LIN {X 0,Y 313.914,Z 800.321,A -85,B 0,C 180,E1 15407.149,E2 15407.149} C_VEL
LIN {X 0,Y 312.972,Z 809.816,A -85,B 0,C 180,E1 15404.241,E2 15404.241} C_VEL
LIN {X 0,Y 312.435,Z 817.558,A -85,B 0,C 180,E1 15401.257,E2 15401.257} C_VEL
LIN {X 0,Y 312.288,Z 823.487,A -85,B 0,C 180,E1 15398.284,E2 15398.284} C_VEL
LIN {X 0,Y 312.342,Z 827.951,A -85,B 0,C 180,E1 15395.143,E2 15395.143} C_VEL
LIN {X 0,Y 312.432,Z 830.624,A -85,B 0,C 180,E1 15392.017,E2 15392.017} C_VEL
LIN {X 0,Y 312.422,Z 831.58,A -85,B 0,C 180,E1 15389.083,E2 15389.083} C_VEL
LIN {X 0,Y 312.275,Z 830.966,A -85,B 0,C 180,E1 15385.961,E2 15385.961} C_VEL
LIN {X 0,Y 312.18,Z 828.719,A -85,B 0,C 180,E1 15382.824,E2 15382.824} C_VEL
LIN {X 0,Y 312.322,Z 824.551,A -85,B 0,C 180,E1 15379.486,E2 15379.486} C_VEL
LIN {X 0,Y 313.004,Z 818.517,A -85,B 0,C 180,E1 15376.138,E2 15376.138} C_VEL
LIN {X 0,Y 314.374,Z 810.506,A -85,B 0,C 180,E1 15372.795,E2 15372.795} C_VEL
LIN {X 0,Y 316.45,Z 800.994,A -85,B 0,C 180,E1 15369.662,E2 15369.662} C_VEL
LIN {X 0,Y 319.412,Z 789.139,A -85,B 0,C 180,E1 15366.517,E2 15366.517} C_VEL
LIN {X 0,Y 322.924,Z 776.215,A -85,B 0,C 180,E1 15363.719,E2 15363.719} C_VEL
LIN {X 0,Y 327.069,Z 761.596,A -85,B 0,C 180,E1 15361.118,E2 15361.118} C_VEL
LIN {X 0,Y 331.687,Z 745.535,A -85,B 0,C 180,E1 15358.769,E2 15358.769} C_VEL
LIN {X 0,Y 336.67,Z 727.913,A -85,B 0,C 180,E1 15356.672,E2 15356.672} C_VEL
LIN {X 0,Y 341.968,Z 708.641,A -85,B 0,C 180,E1 15354.83,E2 15354.83} C_VEL
LIN {X 0,Y 346.988,Z 689.431,A -85,B 0,C 180,E1 15353.382,E2 15353.382} C_VEL
LIN {X 0,Y 351.914,Z 668.887,A -85,B 0,C 180,E1 15352.194,E2 15352.194} C_VEL
LIN {X 0,Y 356.918,Z 643.713,A -85,B 0,C 180,E1 15351.101,E2 15351.101} C_VEL
LIN {X 0,Y 369.381,Z 576.188,A -85,B 0,C 180,E1 15348.561,E2 15348.561} C_VEL
LIN {X 0,Y 384.205,Z 508.645,A -85,B 0,C 180,E1 15346.075,E2 15346.075} C_VEL
LIN {X 0,Y 390.219,Z 483.209,A -85,B 0,C 180,E1 15344.294,E2 15344.294} C_VEL
LIN {X 0,Y 390.2,Z 483.501,A -85,B 0,C 180,E1 15343.942,E2 15343.942} C_VEL
LIN {X 0,Y 372.708,Z 558.454,A -85,B 0,C 180,E1 15341.257,E2 15341.257} C_VEL
LIN {X 0,Y 359.717,Z 624.486,A -85,B 0,C 180,E1 15338.782,E2 15338.782} C_VEL
LIN {X 0,Y 355.652,Z 646.636,A -85,B 0,C 180,E1 15337.785,E2 15337.785} C_VEL
LIN {X 0,Y 351.441,Z 666.051,A -85,B 0,C 180,E1 15336.586,E2 15336.586} C_VEL
LIN {X 0,Y 346.839,Z 684.676,A -85,B 0,C 180,E1 15335.107,E2 15335.107} C_VEL
LIN {X 0,Y 341.835,Z 703.189,A -85,B 0,C 180,E1 15333.259,E2 15333.259} C_VEL
LIN {X 0,Y 336.939,Z 719.84,A -85,B 0,C 180,E1 15331.186,E2 15331.186} C_VEL
LIN {X 0,Y 331.947,Z 735.894,A -85,B 0,C 180,E1 15328.713,E2 15328.713} C_VEL
LIN {X 0,Y 327.477,Z 749.759,A -85,B 0,C 180,E1 15326.082,E2 15326.082} C_VEL
LIN {X 0,Y 323.543,Z 761.616,A -85,B 0,C 180,E1 15323.301,E2 15323.301} C_VEL
LIN {X 0,Y 320.106,Z 771.924,A -85,B 0,C 180,E1 15320.286,E2 15320.286} C_VEL
LIN {X 0,Y 317.4,Z 780.232,A -85,B 0,C 180,E1 15317.224,E2 15317.224} C_VEL
LIN {X 0,Y 315.273,Z 787.058,A -85,B 0,C 180,E1 15313.947,E2 15313.947} C_VEL
LIN {X 0,Y 313.823,Z 792.027,A -85,B 0,C 180,E1 15310.649,E2 15310.649} C_VEL
LIN {X 0,Y 312.936,Z 795.242,A -85,B 0,C 180,E1 15307.342,E2 15307.342} C_VEL
LIN {X 0,Y 312.466,Z 796.765,A -85,B 0,C 180,E1 15304.037,E2 15304.037} C_VEL
LIN {X 0,Y 312.272,Z 796.643,A -85,B 0,C 180,E1 15300.917,E2 15300.917} C_VEL
LIN {X 0,Y 312.209,Z 794.933,A -85,B 0,C 180,E1 15297.704,E2 15297.704} C_VEL
LIN {X 0,Y 312.292,Z 791.564,A -85,B 0,C 180,E1 15294.488,E2 15294.488} C_VEL
LIN {X 0,Y 312.576,Z 786.605,A -85,B 0,C 180,E1 15291.353,E2 15291.353} C_VEL
LIN {X 0,Y 313.171,Z 779.862,A -85,B 0,C 180,E1 15288.209,E2 15288.209} C_VEL
LIN {X 0,Y 314.108,Z 771.702,A -85,B 0,C 180,E1 15285.247,E2 15285.247} C_VEL
LIN {X 0,Y 315.49,Z 761.548,A -85,B 0,C 180,E1 15282.287,E2 15282.287} C_VEL
LIN {X 0,Y 317.239,Z 749.878,A -85,B 0,C 180,E1 15279.522,E2 15279.522} C_VEL
LIN {X 0,Y 319.384,Z 736.161,A -85,B 0,C 180,E1 15276.865,E2 15276.865} C_VEL
LIN {X 0,Y 321.708,Z 721.337,A -85,B 0,C 180,E1 15274.503,E2 15274.503} C_VEL
LIN {X 0,Y 324.195,Z 704.826,A -85,B 0,C 180,E1 15272.344,E2 15272.344} C_VEL
LIN {X 0,Y 326.663,Z 687.236,A -85,B 0,C 180,E1 15270.475,E2 15270.475} C_VEL
LIN {X 0,Y 328.922,Z 669.075,A -85,B 0,C 180,E1 15268.94,E2 15268.94} C_VEL
LIN {X 0,Y 330.927,Z 649.75,A -85,B 0,C 180,E1 15267.67,E2 15267.67} C_VEL
LIN {X 0,Y 332.636,Z 629.153,A -85,B 0,C 180,E1 15266.675,E2 15266.675} C_VEL
LIN {X 0,Y 334.014,Z 605.352,A -85,B 0,C 180,E1 15265.907,E2 15265.907} C_VEL
LIN {X 0,Y 342.851,Z 452.576,A -85,B 0,C 180,E1 15261.576,E2 15261.576} C_VEL
LIN {X 0,Y 328.485,Z 422.487,A -85,B 0,C 180,E1 15259.015,E2 15259.015} C_VEL
LIN {X 0,Y 324.144,Z 413.761,A -85,B 0,C 180,E1 15258.154,E2 15258.154} C_VEL
LIN {X 0,Y 316.77,Z 394.569,A -85,B 0,C 180,E1 15254.74,E2 15254.74} C_VEL
LIN {X 0,Y 314.112,Z 387.671,A -85,B 0,C 180,E1 15253.437,E2 15253.437} C_VEL
LIN {X 0,Y 314.116,Z 387.671,A -85,B 0,C 180,E1 15249.042,E2 15249.042} C_VEL
LIN {X 0,Y 314.129,Z 387.672,A -85,B 0,C 180,E1 15244.733,E2 15244.733} C_VEL
LIN {X 0,Y 314.151,Z 387.67,A -85,B 0,C 180,E1 15240.399,E2 15240.399} C_VEL
LIN {X 0,Y 314.137,Z 387.667,A -85,B 0,C 180,E1 15236.055,E2 15236.055} C_VEL
LIN {X 0,Y 314.122,Z 387.667,A -85,B 0,C 180,E1 15231.651,E2 15231.651} C_VEL
LIN {X 0,Y 314.112,Z 387.664,A -85,B 0,C 180,E1 15227.219,E2 15227.219} C_VEL
LIN {X 0,Y 314.11,Z 387.664,A -85,B 0,C 180,E1 15222.875,E2 15222.875} C_VEL
LIN {X 0,Y 314.128,Z 387.662,A -85,B 0,C 180,E1 15218.419,E2 15218.419} C_VEL
LIN {X 0,Y 314.137,Z 387.66,A -85,B 0,C 180,E1 15214.015,E2 15214.015} C_VEL
LIN {X 0,Y 314.13,Z 387.664,A -85,B 0,C 180,E1 15209.635,E2 15209.635} C_VEL
LIN {X 0,Y 314.112,Z 387.669,A -85,B 0,C 180,E1 15205.253,E2 15205.253} C_VEL
LIN {X 0,Y 314.108,Z 387.668,A -85,B 0,C 180,E1 15200.842,E2 15200.842} C_VEL
LIN {X 0,Y 314.117,Z 387.667,A -85,B 0,C 180,E1 15196.376,E2 15196.376} C_VEL
LIN {X 0,Y 314.133,Z 387.668,A -85,B 0,C 180,E1 15192.016,E2 15192.016} C_VEL
LIN {X 0,Y 314.143,Z 387.669,A -85,B 0,C 180,E1 15187.546,E2 15187.546} C_VEL
LIN {X 0,Y 314.115,Z 387.668,A -85,B 0,C 180,E1 15183.034,E2 15183.034} C_VEL
LIN {X 0,Y 314.109,Z 387.672,A -85,B 0,C 180,E1 15178.531,E2 15178.531} C_VEL
LIN {X 0,Y 314.116,Z 387.676,A -85,B 0,C 180,E1 15174.148,E2 15174.148} C_VEL
LIN {X 0,Y 314.135,Z 387.67,A -85,B 0,C 180,E1 15169.749,E2 15169.749} C_VEL
LIN {X 0,Y 314.134,Z 387.669,A -85,B 0,C 180,E1 15165.297,E2 15165.297} C_VEL
LIN {X 0,Y 313.812,Z 388.707,A -85,B 0,C 180,E1 15164.32,E2 15164.32} C_VEL
LIN {X 0,Y 312.995,Z 391.85,A -85,B 0,C 180,E1 15163.251,E2 15163.251} C_VEL
LIN {X 0,Y 311.72,Z 398.473,A -85,B 0,C 180,E1 15161.831,E2 15161.831} C_VEL
LIN {X 0,Y 311.345,Z 405.44,A -85,B 0,C 180,E1 15160.402,E2 15160.402} C_VEL
LIN {X 0,Y 311.719,Z 407.553,A -85,B 0,C 180,E1 15159.912,E2 15159.912} C_VEL
LIN {X 0,Y 316.265,Z 424.463,A -85,B 0,C 180,E1 15155.968,E2 15155.968} C_VEL
LIN {X 0,Y 319.293,Z 436.92,A -85,B 0,C 180,E1 15153.231,E2 15153.231} C_VEL
LIN {X 0,Y 315.46,Z 463.796,A -85,B 0,C 180,E1 15148.388,E2 15148.388} C_VEL
LIN {X 0,Y 313.788,Z 477.545,A -85,B 0,C 180,E1 15145.985,E2 15145.985} C_VEL
LIN {X 0,Y 317.652,Z 514.782,A -85,B 0,C 180,E1 15144.352,E2 15144.352} C_VEL
LIN {X 0,Y 313.153,Z 610.478,A -85,B 0,C 180,E1 15141.066,E2 15141.066} C_VEL
LIN {X 0,Y 312.346,Z 627.663,A -85,B 0,C 180,E1 15140.142,E2 15140.142} C_VEL
LIN {X 0,Y 311.341,Z 644.035,A -85,B 0,C 180,E1 15138.927,E2 15138.927} C_VEL
LIN {X 0,Y 310.15,Z 660.173,A -85,B 0,C 180,E1 15137.35,E2 15137.35} C_VEL
LIN {X 0,Y 309.02,Z 675.002,A -85,B 0,C 180,E1 15135.482,E2 15135.482} C_VEL
LIN {X 0,Y 307.953,Z 688.503,A -85,B 0,C 180,E1 15133.328,E2 15133.328} C_VEL
LIN {X 0,Y 307.115,Z 699.77,A -85,B 0,C 180,E1 15131.075,E2 15131.075} C_VEL
LIN {X 0,Y 306.548,Z 709.041,A -85,B 0,C 180,E1 15128.776,E2 15128.776} C_VEL
LIN {X 0,Y 306.169,Z 717.713,A -85,B 0,C 180,E1 15125.999,E2 15125.999} C_VEL
LIN {X 0,Y 306.109,Z 723.767,A -85,B 0,C 180,E1 15123.371,E2 15123.371} C_VEL
LIN {X 0,Y 306.331,Z 728.031,A -85,B 0,C 180,E1 15120.748,E2 15120.748} C_VEL
LIN {X 0,Y 306.844,Z 730.658,A -85,B 0,C 180,E1 15117.946,E2 15117.946} C_VEL
LIN {X 0,Y 307.658,Z 731.453,A -85,B 0,C 180,E1 15115.34,E2 15115.34} C_VEL
LIN {X 0,Y 308.807,Z 730.568,A -85,B 0,C 180,E1 15112.746,E2 15112.746} C_VEL
LIN {X 0,Y 310.49,Z 727.787,A -85,B 0,C 180,E1 15109.986,E2 15109.986} C_VEL
LIN {X 0,Y 312.493,Z 723.453,A -85,B 0,C 180,E1 15107.434,E2 15107.434} C_VEL
LIN {X 0,Y 315.283,Z 716.356,A -85,B 0,C 180,E1 15104.598,E2 15104.598} C_VEL
LIN {X 0,Y 318.084,Z 708.328,A -85,B 0,C 180,E1 15102.248,E2 15102.248} C_VEL
LIN {X 0,Y 321.279,Z 698.442,A -85,B 0,C 180,E1 15099.981,E2 15099.981} C_VEL
LIN {X 0,Y 325.031,Z 685.498,A -85,B 0,C 180,E1 15097.672,E2 15097.672} C_VEL
LIN {X 0,Y 328.663,Z 671.745,A -85,B 0,C 180,E1 15095.752,E2 15095.752} C_VEL
LIN {X 0,Y 332.541,Z 655.405,A -85,B 0,C 180,E1 15093.961,E2 15093.961} C_VEL
LIN {X 0,Y 335.996,Z 638.369,A -85,B 0,C 180,E1 15092.532,E2 15092.532} C_VEL
LIN {X 0,Y 338.941,Z 621.261,A -85,B 0,C 180,E1 15091.452,E2 15091.452} C_VEL
LIN {X 0,Y 348.284,Z 567.539,A -85,B 0,C 180,E1 15088.946,E2 15088.946} C_VEL
LIN {X 0,Y 355.162,Z 531.054,A -85,B 0,C 180,E1 15087.337,E2 15087.337} C_VEL
LIN {X 0,Y 355.87,Z 516.287,A -85,B 0,C 180,E1 15085.732,E2 15085.732} C_VEL
LIN {X 0,Y 356.726,Z 501.332,A -85,B 0,C 180,E1 15083.743,E2 15083.743} C_VEL
LIN {X 0,Y 357.866,Z 489.179,A -85,B 0,C 180,E1 15081.767,E2 15081.767} C_VEL
LIN {X 0,Y 357.74,Z 486,A -85,B 0,C 180,E1 15079.731,E2 15079.731} C_VEL
LIN {X 0,Y 358.151,Z 485.015,A -85,B 0,C 180,E1 15078.147,E2 15078.147} C_VEL
LIN {X 0,Y 359.009,Z 484.902,A -85,B 0,C 180,E1 15076.755,E2 15076.755} C_VEL
LIN {X 0,Y 361.058,Z 488.224,A -85,B 0,C 180,E1 15074.401,E2 15074.401} C_VEL
LIN {X 0,Y 361.187,Z 488.98,A -85,B 0,C 180,E1 15074.208,E2 15074.208} C_VEL
LIN {X 0,Y 360.176,Z 501.484,A -85,B 0,C 180,E1 15073.084,E2 15073.084} C_VEL
LIN {X 0,Y 359.266,Z 508.394,A -85,B 0,C 180,E1 15072.71,E2 15072.71} C_VEL
LIN {X 0,Y 347.71,Z 581.363,A -85,B 0,C 180,E1 15070.114,E2 15070.114} C_VEL
LIN {X 0,Y 338.375,Z 654.777,A -85,B 0,C 180,E1 15067.523,E2 15067.523} C_VEL
LIN {X 0,Y 334.909,Z 673.937,A -85,B 0,C 180,E1 15066.556,E2 15066.556} C_VEL
LIN {X 0,Y 330.768,Z 692.92,A -85,B 0,C 180,E1 15065.266,E2 15065.266} C_VEL
LIN {X 0,Y 326.424,Z 710.758,A -85,B 0,C 180,E1 15063.671,E2 15063.671} C_VEL
LIN {X 0,Y 322.018,Z 727.541,A -85,B 0,C 180,E1 15061.756,E2 15061.756} C_VEL
LIN {X 0,Y 317.756,Z 743.428,A -85,B 0,C 180,E1 15059.502,E2 15059.502} C_VEL
LIN {X 0,Y 313.809,Z 758.314,A -85,B 0,C 180,E1 15056.901,E2 15056.901} C_VEL
LIN {X 0,Y 310.363,Z 771.95,A -85,B 0,C 180,E1 15053.949,E2 15053.949} C_VEL
LIN {X 0,Y 308.809,Z 779.29,A -85,B 0,C 180,E1 15052.179,E2 15052.179} C_VEL
LIN {X 0,Y 306.989,Z 791.913,A -85,B 0,C 180,E1 15049.403,E2 15049.403} C_VEL
LIN {X 0,Y 305.657,Z 802.566,A -85,B 0,C 180,E1 15046.535,E2 15046.535} C_VEL
LIN {X 0,Y 304.796,Z 811.742,A -85,B 0,C 180,E1 15043.469,E2 15043.469} C_VEL
LIN {X 0,Y 304.374,Z 818.957,A -85,B 0,C 180,E1 15040.409,E2 15040.409} C_VEL
LIN {X 0,Y 304.315,Z 824.411,A -85,B 0,C 180,E1 15037.362,E2 15037.362} C_VEL
LIN {X 0,Y 304.39,Z 828.204,A -85,B 0,C 180,E1 15034.333,E2 15034.333} C_VEL
LIN {X 0,Y 304.467,Z 830.382,A -85,B 0,C 180,E1 15031.317,E2 15031.317} C_VEL
LIN {X 0,Y 304.405,Z 831.05,A -85,B 0,C 180,E1 15028.306,E2 15028.306} C_VEL
LIN {X 0,Y 304.246,Z 830.152,A -85,B 0,C 180,E1 15025.098,E2 15025.098} C_VEL
LIN {X 0,Y 304.181,Z 827.428,A -85,B 0,C 180,E1 15021.684,E2 15021.684} C_VEL
LIN {X 0,Y 304.497,Z 822.9,A -85,B 0,C 180,E1 15018.253,E2 15018.253} C_VEL
LIN {X 0,Y 305.457,Z 816.503,A -85,B 0,C 180,E1 15014.819,E2 15014.819} C_VEL
LIN {X 0,Y 307.204,Z 808.16,A -85,B 0,C 180,E1 15011.4,E2 15011.4} C_VEL
LIN {X 0,Y 309.712,Z 798.308,A -85,B 0,C 180,E1 15008.206,E2 15008.206} C_VEL
LIN {X 0,Y 313.115,Z 786.372,A -85,B 0,C 180,E1 15005.07,E2 15005.07} C_VEL
LIN {X 0,Y 317.214,Z 772.901,A -85,B 0,C 180,E1 15002.193,E2 15002.193} C_VEL
LIN {X 0,Y 322.052,Z 757.414,A -85,B 0,C 180,E1 14999.495,E2 14999.495} C_VEL
LIN {X 0,Y 327.431,Z 740.36,A -85,B 0,C 180,E1 14997.074,E2 14997.074} C_VEL
LIN {X 0,Y 333.036,Z 722.382,A -85,B 0,C 180,E1 14995.01,E2 14995.01} C_VEL
LIN {X 0,Y 338.673,Z 703.62,A -85,B 0,C 180,E1 14993.285,E2 14993.285} C_VEL
LIN {X 0,Y 344.197,Z 684.057,A -85,B 0,C 180,E1 14991.881,E2 14991.881} C_VEL
LIN {X 0,Y 349.702,Z 662.484,A -85,B 0,C 180,E1 14990.705,E2 14990.705} C_VEL
LIN {X 0,Y 354.983,Z 637.145,A -85,B 0,C 180,E1 14989.648,E2 14989.648} C_VEL
LIN {X 0,Y 369.06,Z 569.328,A -85,B 0,C 180,E1 14987.076,E2 14987.076} C_VEL
LIN {X 0,Y 383.069,Z 510.953,A -85,B 0,C 180,E1 14984.941,E2 14984.941} C_VEL
LIN {X 0,Y 384.903,Z 503.746,A -85,B 0,C 180,E1 14984.433,E2 14984.433} C_VEL
LIN {X 0,Y 366.246,Z 580.486,A -85,B 0,C 180,E1 14981.677,E2 14981.677} C_VEL
LIN {X 0,Y 353.953,Z 639.883,A -85,B 0,C 180,E1 14979.346,E2 14979.346} C_VEL
LIN {X 0,Y 349.545,Z 659.245,A -85,B 0,C 180,E1 14978.264,E2 14978.264} C_VEL
LIN {X 0,Y 344.428,Z 678.747,A -85,B 0,C 180,E1 14976.831,E2 14976.831} C_VEL
LIN {X 0,Y 339.078,Z 697.275,A -85,B 0,C 180,E1 14975.1,E2 14975.1} C_VEL
LIN {X 0,Y 333.777,Z 714.058,A -85,B 0,C 180,E1 14973.14,E2 14973.14} C_VEL
LIN {X 0,Y 328.29,Z 730.451,A -85,B 0,C 180,E1 14970.775,E2 14970.775} C_VEL
LIN {X 0,Y 323.311,Z 744.731,A -85,B 0,C 180,E1 14968.24,E2 14968.24} C_VEL
LIN {X 0,Y 318.706,Z 757.419,A -85,B 0,C 180,E1 14965.455,E2 14965.455} C_VEL
LIN {X 0,Y 314.609,Z 768.541,A -85,B 0,C 180,E1 14962.418,E2 14962.418} C_VEL
LIN {X 0,Y 311.122,Z 778.117,A -85,B 0,C 180,E1 14959.119,E2 14959.119} C_VEL
LIN {X 0,Y 308.492,Z 785.539,A -85,B 0,C 180,E1 14955.798,E2 14955.798} C_VEL
LIN {X 0,Y 306.613,Z 791.116,A -85,B 0,C 180,E1 14952.428,E2 14952.428} C_VEL
LIN {X 0,Y 305.336,Z 795.076,A -85,B 0,C 180,E1 14948.853,E2 14948.853} C_VEL
LIN {X 0,Y 304.656,Z 797.074,A -85,B 0,C 180,E1 14945.461,E2 14945.461} C_VEL
LIN {X 0,Y 304.338,Z 797.395,A -85,B 0,C 180,E1 14942.071,E2 14942.071} C_VEL
LIN {X 0,Y 304.23,Z 796.153,A -85,B 0,C 180,E1 14938.87,E2 14938.87} C_VEL
LIN {X 0,Y 304.248,Z 793.36,A -85,B 0,C 180,E1 14935.665,E2 14935.665} C_VEL
LIN {X 0,Y 304.478,Z 788.598,A -85,B 0,C 180,E1 14932.262,E2 14932.262} C_VEL
LIN {X 0,Y 304.983,Z 782.305,A -85,B 0,C 180,E1 14929.038,E2 14929.038} C_VEL
LIN {X 0,Y 305.824,Z 774.628,A -85,B 0,C 180,E1 14925.999,E2 14925.999} C_VEL
LIN {X 0,Y 307.107,Z 765.001,A -85,B 0,C 180,E1 14922.961,E2 14922.961} C_VEL
LIN {X 0,Y 308.767,Z 753.934,A -85,B 0,C 180,E1 14920.122,E2 14920.122} C_VEL
LIN {X 0,Y 310.92,Z 740.503,A -85,B 0,C 180,E1 14917.3,E2 14917.3} C_VEL
LIN {X 0,Y 313.294,Z 725.893,A -85,B 0,C 180,E1 14914.782,E2 14914.782} C_VEL
LIN {X 0,Y 315.782,Z 710.168,A -85,B 0,C 180,E1 14912.558,E2 14912.558} C_VEL
LIN {X 0,Y 318.316,Z 692.905,A -85,B 0,C 180,E1 14910.574,E2 14910.574} C_VEL
LIN {X 0,Y 320.811,Z 674.138,A -85,B 0,C 180,E1 14908.844,E2 14908.844} C_VEL
LIN {X 0,Y 322.921,Z 655.67,A -85,B 0,C 180,E1 14907.506,E2 14907.506} C_VEL
LIN {X 0,Y 324.788,Z 635.515,A -85,B 0,C 180,E1 14906.402,E2 14906.402} C_VEL
LIN {X 0,Y 326.212,Z 614.334,A -85,B 0,C 180,E1 14905.609,E2 14905.609} C_VEL
LIN {X 0,Y 335.81,Z 455.019,A -85,B 0,C 180,E1 14900.964,E2 14900.964} C_VEL
LIN {X 0,Y 322.329,Z 426.659,A -85,B 0,C 180,E1 14898.482,E2 14898.482} C_VEL
LIN {X 0,Y 316.044,Z 414.082,A -85,B 0,C 180,E1 14897.221,E2 14897.221} C_VEL
LIN {X 0,Y 308.675,Z 395.185,A -85,B 0,C 180,E1 14893.752,E2 14893.752} C_VEL
LIN {X 0,Y 306.203,Z 388.657,A -85,B 0,C 180,E1 14892.526,E2 14892.526} C_VEL
LIN {X 0,Y 306.198,Z 388.656,A -85,B 0,C 180,E1 14888.097,E2 14888.097} C_VEL
LIN {X 0,Y 306.179,Z 388.661,A -85,B 0,C 180,E1 14883.619,E2 14883.619} C_VEL
LIN {X 0,Y 306.172,Z 388.657,A -85,B 0,C 180,E1 14879.117,E2 14879.117} C_VEL
LIN {X 0,Y 306.187,Z 388.658,A -85,B 0,C 180,E1 14874.708,E2 14874.708} C_VEL
LIN {X 0,Y 306.204,Z 388.653,A -85,B 0,C 180,E1 14870.251,E2 14870.251} C_VEL
LIN {X 0,Y 306.188,Z 388.661,A -85,B 0,C 180,E1 14865.726,E2 14865.726} C_VEL
LIN {X 0,Y 306.173,Z 388.66,A -85,B 0,C 180,E1 14861.3,E2 14861.3} C_VEL
LIN {X 0,Y 306.175,Z 388.657,A -85,B 0,C 180,E1 14856.752,E2 14856.752} C_VEL
LIN {X 0,Y 306.192,Z 388.652,A -85,B 0,C 180,E1 14852.236,E2 14852.236} C_VEL
LIN {X 0,Y 306.199,Z 388.646,A -85,B 0,C 180,E1 14847.941,E2 14847.941} C_VEL
LIN {X 0,Y 306.182,Z 388.653,A -85,B 0,C 180,E1 14843.437,E2 14843.437} C_VEL
LIN {X 0,Y 306.17,Z 388.658,A -85,B 0,C 180,E1 14838.891,E2 14838.891} C_VEL
LIN {X 0,Y 306.173,Z 388.661,A -85,B 0,C 180,E1 14834.446,E2 14834.446} C_VEL
LIN {X 0,Y 306.197,Z 388.658,A -85,B 0,C 180,E1 14829.948,E2 14829.948} C_VEL
LIN {X 0,Y 306.196,Z 388.655,A -85,B 0,C 180,E1 14825.499,E2 14825.499} C_VEL
LIN {X 0,Y 306.179,Z 388.657,A -85,B 0,C 180,E1 14821.067,E2 14821.067} C_VEL
LIN {X 0,Y 306.17,Z 388.664,A -85,B 0,C 180,E1 14816.502,E2 14816.502} C_VEL
LIN {X 0,Y 306.176,Z 388.664,A -85,B 0,C 180,E1 14812.125,E2 14812.125} C_VEL
LIN {X 0,Y 306.197,Z 388.658,A -85,B 0,C 180,E1 14807.726,E2 14807.726} C_VEL
LIN {X 0,Y 306.196,Z 388.85,A -85,B 0,C 180,E1 14804.613,E2 14804.613} C_VEL
LIN {X 0,Y 311.185,Z 405.516,A -85,B 0,C 180,E1 14800.403,E2 14800.403} C_VEL
LIN {X 0,Y 311.719,Z 407.553,A -85,B 0,C 180,E1 14799.912,E2 14799.912} C_VEL
LIN {X 0,Y 312.041,Z 412.58,A -85,B 0,C 180,E1 14798.827,E2 14798.827} C_VEL
LIN {X 0,Y 309.592,Z 428.14,A -85,B 0,C 180,E1 14795.884,E2 14795.884} C_VEL
LIN {X 0,Y 309.952,Z 431.807,A -85,B 0,C 180,E1 14795.106,E2 14795.106} C_VEL
LIN {X 0,Y 311.591,Z 439.271,A -85,B 0,C 180,E1 14793.455,E2 14793.455} C_VEL
LIN {X 0,Y 307.589,Z 466.366,A -85,B 0,C 180,E1 14788.478,E2 14788.478} C_VEL
LIN {X 0,Y 306.18,Z 477.362,A -85,B 0,C 180,E1 14786.52,E2 14786.52} C_VEL
LIN {X 0,Y 310.041,Z 515.528,A -85,B 0,C 180,E1 14784.8,E2 14784.8} C_VEL
LIN {X 0,Y 305.377,Z 611.092,A -85,B 0,C 180,E1 14781.406,E2 14781.406} C_VEL
LIN {X 0,Y 304.546,Z 628.058,A -85,B 0,C 180,E1 14780.466,E2 14780.466} C_VEL
LIN {X 0,Y 303.441,Z 645.323,A -85,B 0,C 180,E1 14779.139,E2 14779.139} C_VEL
LIN {X 0,Y 302.217,Z 661.31,A -85,B 0,C 180,E1 14777.522,E2 14777.522} C_VEL
LIN {X 0,Y 301.013,Z 676.765,A -85,B 0,C 180,E1 14775.509,E2 14775.509} C_VEL
LIN {X 0,Y 299.899,Z 690.654,A -85,B 0,C 180,E1 14773.212,E2 14773.212} C_VEL
LIN {X 0,Y 299.048,Z 702.238,A -85,B 0,C 180,E1 14770.792,E2 14770.792} C_VEL
LIN {X 0,Y 298.478,Z 711.743,A -85,B 0,C 180,E1 14768.282,E2 14768.282} C_VEL
LIN {X 0,Y 298.191,Z 719.199,A -85,B 0,C 180,E1 14765.774,E2 14765.774} C_VEL
LIN {X 0,Y 298.179,Z 725.59,A -85,B 0,C 180,E1 14762.883,E2 14762.883} C_VEL
LIN {X 0,Y 298.46,Z 729.696,A -85,B 0,C 180,E1 14760.192,E2 14760.192} C_VEL
LIN {X 0,Y 299.104,Z 732.227,A -85,B 0,C 180,E1 14757.318,E2 14757.318} C_VEL
LIN {X 0,Y 300.046,Z 732.895,A -85,B 0,C 180,E1 14754.646,E2 14754.646} C_VEL
LIN {X 0,Y 301.605,Z 731.64,A -85,B 0,C 180,E1 14751.613,E2 14751.613} C_VEL
LIN {X 0,Y 303.429,Z 728.808,A -85,B 0,C 180,E1 14748.982,E2 14748.982} C_VEL
LIN {X 0,Y 306.068,Z 723.475,A -85,B 0,C 180,E1 14746.011,E2 14746.011} C_VEL
LIN {X 0,Y 308.888,Z 716.782,A -85,B 0,C 180,E1 14743.45,E2 14743.45} C_VEL
LIN {X 0,Y 312.242,Z 708.123,A -85,B 0,C 180,E1 14740.936,E2 14740.936} C_VEL
LIN {X 0,Y 316.092,Z 697.002,A -85,B 0,C 180,E1 14738.474,E2 14738.474} C_VEL
LIN {X 0,Y 319.791,Z 685.109,A -85,B 0,C 180,E1 14736.409,E2 14736.409} C_VEL
LIN {X 0,Y 323.633,Z 671.93,A -85,B 0,C 180,E1 14734.568,E2 14734.568} C_VEL
LIN {X 0,Y 327.842,Z 655.543,A -85,B 0,C 180,E1 14732.776,E2 14732.776} C_VEL
LIN {X 0,Y 331.607,Z 638.669,A -85,B 0,C 180,E1 14731.353,E2 14731.353} C_VEL
LIN {X 0,Y 334.979,Z 620.426,A -85,B 0,C 180,E1 14730.212,E2 14730.212} C_VEL
LIN {X 0,Y 349.202,Z 546.392,A -85,B 0,C 180,E1 14726.798,E2 14726.798} C_VEL
LIN {X 0,Y 351.782,Z 533.481,A -85,B 0,C 180,E1 14726.207,E2 14726.207} C_VEL
LIN {X 0,Y 352.944,Z 518.858,A -85,B 0,C 180,E1 14724.547,E2 14724.547} C_VEL
LIN {X 0,Y 354.336,Z 504.754,A -85,B 0,C 180,E1 14722.574,E2 14722.574} C_VEL
LIN {X 0,Y 355.578,Z 495.959,A -85,B 0,C 180,E1 14721.115,E2 14721.115} C_VEL
LIN {X 0,Y 355.805,Z 493.186,A -85,B 0,C 180,E1 14719.099,E2 14719.099} C_VEL
LIN {X 0,Y 356.921,Z 492.592,A -85,B 0,C 180,E1 14716.88,E2 14716.88} C_VEL
LIN {X 0,Y 358.347,Z 495.123,A -85,B 0,C 180,E1 14715.013,E2 14715.013} C_VEL
LIN {X 0,Y 357.154,Z 505.327,A -85,B 0,C 180,E1 14714.124,E2 14714.124} C_VEL
LIN {X 0,Y 356.168,Z 511.22,A -85,B 0,C 180,E1 14713.837,E2 14713.837} C_VEL
LIN {X 0,Y 343.538,Z 584.251,A -85,B 0,C 180,E1 14711.193,E2 14711.193} C_VEL
LIN {X 0,Y 333.743,Z 653.597,A -85,B 0,C 180,E1 14708.67,E2 14708.67} C_VEL
LIN {X 0,Y 330.101,Z 672.207,A -85,B 0,C 180,E1 14707.724,E2 14707.724} C_VEL
LIN {X 0,Y 325.437,Z 691.939,A -85,B 0,C 180,E1 14706.368,E2 14706.368} C_VEL
LIN {X 0,Y 320.808,Z 709.452,A -85,B 0,C 180,E1 14704.775,E2 14704.775} C_VEL
LIN {X 0,Y 316.066,Z 726.027,A -85,B 0,C 180,E1 14702.856,E2 14702.856} C_VEL
LIN {X 0,Y 311.448,Z 741.786,A -85,B 0,C 180,E1 14700.587,E2 14700.587} C_VEL
LIN {X 0,Y 307.127,Z 756.577,A -85,B 0,C 180,E1 14697.956,E2 14697.956} C_VEL
LIN {X 0,Y 303.325,Z 770.18,A -85,B 0,C 180,E1 14694.957,E2 14694.957} C_VEL
LIN {X 0,Y 300.379,Z 782.453,A -85,B 0,C 180,E1 14691.684,E2 14691.684} C_VEL
LIN {X 0,Y 298.602,Z 794.732,A -85,B 0,C 180,E1 14688.751,E2 14688.751} C_VEL
LIN {X 0,Y 297.401,Z 804.799,A -85,B 0,C 180,E1 14685.803,E2 14685.803} C_VEL
LIN {X 0,Y 296.653,Z 813.434,A -85,B 0,C 180,E1 14682.655,E2 14682.655} C_VEL
LIN {X 0,Y 296.349,Z 820.143,A -85,B 0,C 180,E1 14679.516,E2 14679.516} C_VEL
LIN {X 0,Y 296.359,Z 825.103,A -85,B 0,C 180,E1 14676.392,E2 14676.392} C_VEL
LIN {X 0,Y 296.45,Z 828.421,A -85,B 0,C 180,E1 14673.287,E2 14673.287} C_VEL
LIN {X 0,Y 296.491,Z 830.183,A -85,B 0,C 180,E1 14670.193,E2 14670.193} C_VEL
LIN {X 0,Y 296.353,Z 830.433,A -85,B 0,C 180,E1 14667.039,E2 14667.039} C_VEL
LIN {X 0,Y 296.195,Z 829.114,A -85,B 0,C 180,E1 14663.799,E2 14663.799} C_VEL
LIN {X 0,Y 296.253,Z 825.872,A -85,B 0,C 180,E1 14660.232,E2 14660.232} C_VEL
LIN {X 0,Y 296.886,Z 820.612,A -85,B 0,C 180,E1 14656.563,E2 14656.563} C_VEL
LIN {X 0,Y 298.255,Z 813.667,A -85,B 0,C 180,E1 14653.043,E2 14653.043} C_VEL
LIN {X 0,Y 300.54,Z 804.744,A -85,B 0,C 180,E1 14649.554,E2 14649.554} C_VEL
LIN {X 0,Y 303.712,Z 794.08,A -85,B 0,C 180,E1 14646.235,E2 14646.235} C_VEL
LIN {X 0,Y 307.959,Z 781.042,A -85,B 0,C 180,E1 14642.964,E2 14642.964} C_VEL
LIN {X 0,Y 312.801,Z 766.923,A -85,B 0,C 180,E1 14640.089,E2 14640.089} C_VEL
LIN {X 0,Y 318.227,Z 751.381,A -85,B 0,C 180,E1 14637.501,E2 14637.501} C_VEL
LIN {X 0,Y 324.126,Z 734.36,A -85,B 0,C 180,E1 14635.202,E2 14635.202} C_VEL
LIN {X 0,Y 330.671,Z 715.08,A -85,B 0,C 180,E1 14633.115,E2 14633.115} C_VEL
LIN {X 0,Y 336.995,Z 695.67,A -85,B 0,C 180,E1 14631.459,E2 14631.459} C_VEL
LIN {X 0,Y 343.157,Z 675.254,A -85,B 0,C 180,E1 14630.132,E2 14630.132} C_VEL
LIN {X 0,Y 349.311,Z 651.833,A -85,B 0,C 180,E1 14628.989,E2 14628.989} C_VEL
LIN {X 0,Y 368.435,Z 567.445,A -85,B 0,C 180,E1 14625.75,E2 14625.75} C_VEL
LIN {X 0,Y 376.625,Z 535.288,A -85,B 0,C 180,E1 14624.574,E2 14624.574} C_VEL
LIN {X 0,Y 358.521,Z 608.198,A -85,B 0,C 180,E1 14621.894,E2 14621.894} C_VEL
LIN {X 0,Y 351.013,Z 642.237,A -85,B 0,C 180,E1 14620.5,E2 14620.5} C_VEL
LIN {X 0,Y 345.977,Z 661.832,A -85,B 0,C 180,E1 14619.371,E2 14619.371} C_VEL
LIN {X 0,Y 340.257,Z 681.365,A -85,B 0,C 180,E1 14617.89,E2 14617.89} C_VEL
LIN {X 0,Y 334.524,Z 699.102,A -85,B 0,C 180,E1 14616.179,E2 14616.179} C_VEL
LIN {X 0,Y 328.403,Z 716.563,A -85,B 0,C 180,E1 14614.07,E2 14614.07} C_VEL
LIN {X 0,Y 322.545,Z 732.421,A -85,B 0,C 180,E1 14611.697,E2 14611.697} C_VEL
LIN {X 0,Y 317.023,Z 746.687,A -85,B 0,C 180,E1 14609.058,E2 14609.058} C_VEL
LIN {X 0,Y 312.02,Z 759.16,A -85,B 0,C 180,E1 14606.2,E2 14606.2} C_VEL
LIN {X 0,Y 307.442,Z 770.461,A -85,B 0,C 180,E1 14602.971,E2 14602.971} C_VEL
LIN {X 0,Y 303.727,Z 779.682,A -85,B 0,C 180,E1 14599.62,E2 14599.62} C_VEL
LIN {X 0,Y 300.845,Z 786.958,A -85,B 0,C 180,E1 14596.158,E2 14596.158} C_VEL
LIN {X 0,Y 298.747,Z 792.416,A -85,B 0,C 180,E1 14592.565,E2 14592.565} C_VEL
LIN {X 0,Y 297.448,Z 795.909,A -85,B 0,C 180,E1 14589.09,E2 14589.09} C_VEL
LIN {X 0,Y 296.704,Z 797.726,A -85,B 0,C 180,E1 14585.608,E2 14585.608} C_VEL
LIN {X 0,Y 296.367,Z 797.921,A -85,B 0,C 180,E1 14582.32,E2 14582.32} C_VEL
LIN {X 0,Y 296.242,Z 796.605,A -85,B 0,C 180,E1 14579.033,E2 14579.033} C_VEL
LIN {X 0,Y 296.25,Z 793.741,A -85,B 0,C 180,E1 14575.742,E2 14575.742} C_VEL
LIN {X 0,Y 296.462,Z 789.232,A -85,B 0,C 180,E1 14572.442,E2 14572.442} C_VEL
LIN {X 0,Y 296.964,Z 782.96,A -85,B 0,C 180,E1 14569.132,E2 14569.132} C_VEL
LIN {X 0,Y 297.818,Z 775.247,A -85,B 0,C 180,E1 14565.992,E2 14565.992} C_VEL
LIN {X 0,Y 299.114,Z 765.687,A -85,B 0,C 180,E1 14562.892,E2 14562.892} C_VEL
LIN {X 0,Y 300.81,Z 754.638,A -85,B 0,C 180,E1 14559.979,E2 14559.979} C_VEL
LIN {X 0,Y 303.016,Z 741.227,A -85,B 0,C 180,E1 14557.085,E2 14557.085} C_VEL
LIN {X 0,Y 305.452,Z 726.646,A -85,B 0,C 180,E1 14554.504,E2 14554.504} C_VEL
LIN {X 0,Y 307.998,Z 711.062,A -85,B 0,C 180,E1 14552.235,E2 14552.235} C_VEL
LIN {X 0,Y 310.637,Z 693.659,A -85,B 0,C 180,E1 14550.178,E2 14550.178} C_VEL
LIN {X 0,Y 313.176,Z 675.187,A -85,B 0,C 180,E1 14548.426,E2 14548.426} C_VEL
LIN {X 0,Y 315.419,Z 656.255,A -85,B 0,C 180,E1 14547.014,E2 14547.014} C_VEL
LIN {X 0,Y 317.35,Z 636.177,A -85,B 0,C 180,E1 14545.881,E2 14545.881} C_VEL
LIN {X 0,Y 318.843,Z 615.029,A -85,B 0,C 180,E1 14545.061,E2 14545.061} C_VEL
LIN {X 0,Y 328.799,Z 457.39,A -85,B 0,C 180,E1 14540.331,E2 14540.331} C_VEL
LIN {X 0,Y 315.617,Z 429.781,A -85,B 0,C 180,E1 14537.843,E2 14537.843} C_VEL
LIN {X 0,Y 307.98,Z 414.46,A -85,B 0,C 180,E1 14536.25,E2 14536.25} C_VEL
LIN {X 0,Y 300.587,Z 395.866,A -85,B 0,C 180,E1 14532.733,E2 14532.733} C_VEL
LIN {X 0,Y 298.237,Z 389.647,A -85,B 0,C 180,E1 14531.494,E2 14531.494} C_VEL
LIN {X 0,Y 298.246,Z 389.65,A -85,B 0,C 180,E1 14526.877,E2 14526.877} C_VEL
LIN {X 0,Y 298.267,Z 389.646,A -85,B 0,C 180,E1 14522.353,E2 14522.353} C_VEL
LIN {X 0,Y 298.249,Z 389.647,A -85,B 0,C 180,E1 14517.774,E2 14517.774} C_VEL
LIN {X 0,Y 298.235,Z 389.646,A -85,B 0,C 180,E1 14513.095,E2 14513.095} C_VEL
LIN {X 0,Y 298.25,Z 389.648,A -85,B 0,C 180,E1 14508.571,E2 14508.571} C_VEL
LIN {X 0,Y 298.266,Z 389.642,A -85,B 0,C 180,E1 14503.967,E2 14503.967} C_VEL
LIN {X 0,Y 298.238,Z 389.642,A -85,B 0,C 180,E1 14499.455,E2 14499.455} C_VEL
LIN {X 0,Y 298.234,Z 389.644,A -85,B 0,C 180,E1 14494.808,E2 14494.808} C_VEL
LIN {X 0,Y 298.257,Z 389.647,A -85,B 0,C 180,E1 14490.192,E2 14490.192} C_VEL
LIN {X 0,Y 298.247,Z 389.647,A -85,B 0,C 180,E1 14485.578,E2 14485.578} C_VEL
LIN {X 0,Y 298.234,Z 389.646,A -85,B 0,C 180,E1 14481.128,E2 14481.128} C_VEL
LIN {X 0,Y 298.237,Z 389.645,A -85,B 0,C 180,E1 14476.427,E2 14476.427} C_VEL
LIN {X 0,Y 298.264,Z 389.646,A -85,B 0,C 180,E1 14471.834,E2 14471.834} C_VEL
LIN {X 0,Y 298.243,Z 389.647,A -85,B 0,C 180,E1 14467.212,E2 14467.212} C_VEL
LIN {X 0,Y 298.233,Z 389.646,A -85,B 0,C 180,E1 14462.657,E2 14462.657} C_VEL
LIN {X 0,Y 298.239,Z 389.65,A -85,B 0,C 180,E1 14458.241,E2 14458.241} C_VEL
LIN {X 0,Y 298.252,Z 389.651,A -85,B 0,C 180,E1 14453.841,E2 14453.841} C_VEL
LIN {X 0,Y 298.257,Z 389.649,A -85,B 0,C 180,E1 14449.256,E2 14449.256} C_VEL
LIN {X 0,Y 298.279,Z 389.811,A -85,B 0,C 180,E1 14445.458,E2 14445.458} C_VEL
LIN {X 0,Y 303.24,Z 406.512,A -85,B 0,C 180,E1 14441.112,E2 14441.112} C_VEL
LIN {X 0,Y 307.682,Z 422.71,A -85,B 0,C 180,E1 14437.189,E2 14437.189} C_VEL
LIN {X 0,Y 309.952,Z 431.807,A -85,B 0,C 180,E1 14435.106,E2 14435.106} C_VEL
LIN {X 0,Y 310.039,Z 435.512,A -85,B 0,C 180,E1 14434.354,E2 14434.354} C_VEL
LIN {X 0,Y 308.356,Z 441.08,A -85,B 0,C 180,E1 14433.393,E2 14433.393} C_VEL
LIN {X 0,Y 302.197,Z 454.23,A -85,B 0,C 180,E1 14431.291,E2 14431.291} C_VEL
LIN {X 0,Y 301.345,Z 457.514,A -85,B 0,C 180,E1 14430.704,E2 14430.704} C_VEL
LIN {X 0,Y 298.591,Z 477.196,A -85,B 0,C 180,E1 14427.073,E2 14427.073} C_VEL
LIN {X 0,Y 302.431,Z 516.309,A -85,B 0,C 180,E1 14425.258,E2 14425.258} C_VEL
LIN {X 0,Y 297.598,Z 611.133,A -85,B 0,C 180,E1 14421.761,E2 14421.761} C_VEL
LIN {X 0,Y 296.718,Z 628.599,A -85,B 0,C 180,E1 14420.773,E2 14420.773} C_VEL
LIN {X 0,Y 295.618,Z 645.403,A -85,B 0,C 180,E1 14419.461,E2 14419.461} C_VEL
LIN {X 0,Y 294.355,Z 661.576,A -85,B 0,C 180,E1 14417.801,E2 14417.801} C_VEL
LIN {X 0,Y 293.111,Z 677.223,A -85,B 0,C 180,E1 14415.735,E2 14415.735} C_VEL
LIN {X 0,Y 291.958,Z 691.327,A -85,B 0,C 180,E1 14413.366,E2 14413.366} C_VEL
LIN {X 0,Y 291.037,Z 703.668,A -85,B 0,C 180,E1 14410.716,E2 14410.716} C_VEL
LIN {X 0,Y 290.442,Z 713.849,A -85,B 0,C 180,E1 14407.915,E2 14407.915} C_VEL
LIN {X 0,Y 290.195,Z 721.239,A -85,B 0,C 180,E1 14405.286,E2 14405.286} C_VEL
LIN {X 0,Y 290.25,Z 727.077,A -85,B 0,C 180,E1 14402.555,E2 14402.555} C_VEL
LIN {X 0,Y 290.587,Z 731.128,A -85,B 0,C 180,E1 14399.803,E2 14399.803} C_VEL
LIN {X 0,Y 291.325,Z 733.685,A -85,B 0,C 180,E1 14396.852,E2 14396.852} C_VEL
LIN {X 0,Y 292.394,Z 734.36,A -85,B 0,C 180,E1 14394.112,E2 14394.112} C_VEL
LIN {X 0,Y 294.015,Z 733.282,A -85,B 0,C 180,E1 14391.198,E2 14391.198} C_VEL
LIN {X 0,Y 296.16,Z 730.38,A -85,B 0,C 180,E1 14388.313,E2 14388.313} C_VEL
LIN {X 0,Y 298.858,Z 725.508,A -85,B 0,C 180,E1 14385.468,E2 14385.468} C_VEL
LIN {X 0,Y 301.926,Z 719.153,A -85,B 0,C 180,E1 14382.859,E2 14382.859} C_VEL
LIN {X 0,Y 305.794,Z 710.103,A -85,B 0,C 180,E1 14380.12,E2 14380.12} C_VEL
LIN {X 0,Y 309.628,Z 700.076,A -85,B 0,C 180,E1 14377.801,E2 14377.801} C_VEL
LIN {X 0,Y 313.794,Z 688.332,A -85,B 0,C 180,E1 14375.63,E2 14375.63} C_VEL
LIN {X 0,Y 318.456,Z 673.751,A -85,B 0,C 180,E1 14373.523,E2 14373.523} C_VEL
LIN {X 0,Y 322.996,Z 657.845,A -85,B 0,C 180,E1 14371.73,E2 14371.73} C_VEL
LIN {X 0,Y 327.257,Z 640.565,A -85,B 0,C 180,E1 14370.233,E2 14370.233} C_VEL
LIN {X 0,Y 330.955,Z 622.49,A -85,B 0,C 180,E1 14369.072,E2 14369.072} C_VEL
LIN {X 0,Y 343.879,Z 558.825,A -85,B 0,C 180,E1 14366.077,E2 14366.077} C_VEL
LIN {X 0,Y 348.777,Z 536.172,A -85,B 0,C 180,E1 14365.061,E2 14365.061} C_VEL
LIN {X 0,Y 350.5,Z 521.327,A -85,B 0,C 180,E1 14363.299,E2 14363.299} C_VEL
LIN {X 0,Y 352.519,Z 507.439,A -85,B 0,C 180,E1 14361.26,E2 14361.26} C_VEL
LIN {X 0,Y 353.426,Z 502.848,A -85,B 0,C 180,E1 14360.466,E2 14360.466} C_VEL
LIN {X 0,Y 353.881,Z 500.735,A -85,B 0,C 180,E1 14358.726,E2 14358.726} C_VEL
LIN {X 0,Y 354.907,Z 500.443,A -85,B 0,C 180,E1 14356.859,E2 14356.859} C_VEL
LIN {X 0,Y 355.583,Z 502.055,A -85,B 0,C 180,E1 14355.771,E2 14355.771} C_VEL
LIN {X 0,Y 354.454,Z 509.256,A -85,B 0,C 180,E1 14355.19,E2 14355.19} C_VEL
LIN {X 0,Y 341.327,Z 577.697,A -85,B 0,C 180,E1 14352.668,E2 14352.668} C_VEL
LIN {X 0,Y 329.45,Z 652.615,A -85,B 0,C 180,E1 14349.869,E2 14349.869} C_VEL
LIN {X 0,Y 325.509,Z 671.13,A -85,B 0,C 180,E1 14348.915,E2 14348.915} C_VEL
LIN {X 0,Y 320.294,Z 691.441,A -85,B 0,C 180,E1 14347.498,E2 14347.498} C_VEL
LIN {X 0,Y 315.13,Z 709.264,A -85,B 0,C 180,E1 14345.831,E2 14345.831} C_VEL
LIN {X 0,Y 309.845,Z 726.224,A -85,B 0,C 180,E1 14343.806,E2 14343.806} C_VEL
LIN {X 0,Y 304.883,Z 741.679,A -85,B 0,C 180,E1 14341.498,E2 14341.498} C_VEL
LIN {X 0,Y 300.305,Z 755.934,A -85,B 0,C 180,E1 14338.867,E2 14338.867} C_VEL
LIN {X 0,Y 296.17,Z 769.285,A -85,B 0,C 180,E1 14335.817,E2 14335.817} C_VEL
LIN {X 0,Y 292.906,Z 781.122,A -85,B 0,C 180,E1 14332.478,E2 14332.478} C_VEL
LIN {X 0,Y 291.904,Z 785.78,A -85,B 0,C 180,E1 14331.079,E2 14331.079} C_VEL
LIN {X 0,Y 290.238,Z 797.434,A -85,B 0,C 180,E1 14328.046,E2 14328.046} C_VEL
LIN {X 0,Y 289.175,Z 806.876,A -85,B 0,C 180,E1 14325.03,E2 14325.03} C_VEL
LIN {X 0,Y 288.539,Z 814.958,A -85,B 0,C 180,E1 14321.797,E2 14321.797} C_VEL
LIN {X 0,Y 288.351,Z 821.18,A -85,B 0,C 180,E1 14318.575,E2 14318.575} C_VEL
LIN {X 0,Y 288.411,Z 825.691,A -85,B 0,C 180,E1 14315.371,E2 14315.371} C_VEL
LIN {X 0,Y 288.503,Z 828.578,A -85,B 0,C 180,E1 14312.185,E2 14312.185} C_VEL
LIN {X 0,Y 288.48,Z 829.865,A -85,B 0,C 180,E1 14309.007,E2 14309.007} C_VEL
LIN {X 0,Y 288.299,Z 829.663,A -85,B 0,C 180,E1 14305.823,E2 14305.823} C_VEL
LIN {X 0,Y 288.178,Z 827.882,A -85,B 0,C 180,E1 14302.424,E2 14302.424} C_VEL
LIN {X 0,Y 288.406,Z 824.273,A -85,B 0,C 180,E1 14298.805,E2 14298.805} C_VEL
LIN {X 0,Y 289.397,Z 818.521,A -85,B 0,C 180,E1 14294.982,E2 14294.982} C_VEL
LIN {X 0,Y 291.214,Z 811.173,A -85,B 0,C 180,E1 14291.373,E2 14291.373} C_VEL
LIN {X 0,Y 294.046,Z 801.88,A -85,B 0,C 180,E1 14287.825,E2 14287.825} C_VEL
LIN {X 0,Y 297.969,Z 790.476,A -85,B 0,C 180,E1 14284.35,E2 14284.35} C_VEL
LIN {X 0,Y 302.75,Z 777.495,A -85,B 0,C 180,E1 14281.172,E2 14281.172} C_VEL
LIN {X 0,Y 308.244,Z 763.05,A -85,B 0,C 180,E1 14278.299,E2 14278.299} C_VEL
LIN {X 0,Y 314.512,Z 746.779,A -85,B 0,C 180,E1 14275.668,E2 14275.668} C_VEL
LIN {X 0,Y 321.419,Z 728.793,A -85,B 0,C 180,E1 14273.325,E2 14273.325} C_VEL
LIN {X 0,Y 328.412,Z 710.026,A -85,B 0,C 180,E1 14271.381,E2 14271.381} C_VEL
LIN {X 0,Y 335.376,Z 690.299,A -85,B 0,C 180,E1 14269.8,E2 14269.8} C_VEL
LIN {X 0,Y 342.071,Z 669.646,A -85,B 0,C 180,E1 14268.543,E2 14268.543} C_VEL
LIN {X 0,Y 348.494,Z 646.546,A -85,B 0,C 180,E1 14267.48,E2 14267.48} C_VEL
LIN {X 0,Y 367.202,Z 570.701,A -85,B 0,C 180,E1 14264.579,E2 14264.579} C_VEL
LIN {X 0,Y 349.512,Z 640.958,A -85,B 0,C 180,E1 14261.87,E2 14261.87} C_VEL
LIN {X 0,Y 344.244,Z 660.179,A -85,B 0,C 180,E1 14260.807,E2 14260.807} C_VEL
LIN {X 0,Y 338.301,Z 678.737,A -85,B 0,C 180,E1 14259.452,E2 14259.452} C_VEL
LIN {X 0,Y 331.497,Z 697.944,A -85,B 0,C 180,E1 14257.646,E2 14257.646} C_VEL
LIN {X 0,Y 325.063,Z 714.766,A -85,B 0,C 180,E1 14255.653,E2 14255.653} C_VEL
LIN {X 0,Y 318.386,Z 731.147,A -85,B 0,C 180,E1 14253.23,E2 14253.23} C_VEL
LIN {X 0,Y 312.299,Z 745.507,A -85,B 0,C 180,E1 14250.601,E2 14250.601} C_VEL
LIN {X 0,Y 306.826,Z 758.022,A -85,B 0,C 180,E1 14247.775,E2 14247.775} C_VEL
LIN {X 0,Y 301.863,Z 769.049,A -85,B 0,C 180,E1 14244.667,E2 14244.667} C_VEL
LIN {X 0,Y 297.781,Z 778.097,A -85,B 0,C 180,E1 14241.468,E2 14241.468} C_VEL
LIN {X 0,Y 294.204,Z 786.078,A -85,B 0,C 180,E1 14237.81,E2 14237.81} C_VEL
LIN {X 0,Y 291.723,Z 791.757,A -85,B 0,C 180,E1 14234.287,E2 14234.287} C_VEL
LIN {X 0,Y 290.034,Z 795.695,A -85,B 0,C 180,E1 14230.728,E2 14230.728} C_VEL
LIN {X 0,Y 289.012,Z 797.96,A -85,B 0,C 180,E1 14227.154,E2 14227.154} C_VEL
LIN {X 0,Y 288.483,Z 798.573,A -85,B 0,C 180,E1 14223.577,E2 14223.577} C_VEL
LIN {X 0,Y 288.278,Z 797.603,A -85,B 0,C 180,E1 14220.198,E2 14220.198} C_VEL
LIN {X 0,Y 288.236,Z 795.003,A -85,B 0,C 180,E1 14216.707,E2 14216.707} C_VEL
LIN {X 0,Y 288.387,Z 790.72,A -85,B 0,C 180,E1 14213.23,E2 14213.23} C_VEL
LIN {X 0,Y 288.824,Z 784.796,A -85,B 0,C 180,E1 14209.831,E2 14209.831} C_VEL
LIN {X 0,Y 289.663,Z 776.981,A -85,B 0,C 180,E1 14206.424,E2 14206.424} C_VEL
LIN {X 0,Y 290.926,Z 767.664,A -85,B 0,C 180,E1 14203.22,E2 14203.22} C_VEL
LIN {X 0,Y 292.594,Z 756.915,A -85,B 0,C 180,E1 14200.226,E2 14200.226} C_VEL
LIN {X 0,Y 294.78,Z 743.831,A -85,B 0,C 180,E1 14197.252,E2 14197.252} C_VEL
LIN {X 0,Y 297.214,Z 729.633,A -85,B 0,C 180,E1 14194.6,E2 14194.6} C_VEL
LIN {X 0,Y 299.88,Z 713.831,A -85,B 0,C 180,E1 14192.174,E2 14192.174} C_VEL
LIN {X 0,Y 302.555,Z 697.042,A -85,B 0,C 180,E1 14190.065,E2 14190.065} C_VEL
LIN {X 0,Y 305.132,Z 679.344,A -85,B 0,C 180,E1 14188.269,E2 14188.269} C_VEL
LIN {X 0,Y 307.533,Z 660.2,A -85,B 0,C 180,E1 14186.741,E2 14186.741} C_VEL
LIN {X 0,Y 309.648,Z 639.518,A -85,B 0,C 180,E1 14185.49,E2 14185.49} C_VEL
LIN {X 0,Y 311.266,Z 618.954,A -85,B 0,C 180,E1 14184.612,E2 14184.612} C_VEL
LIN {X 0,Y 321.733,Z 459.657,A -85,B 0,C 180,E1 14179.668,E2 14179.668} C_VEL
LIN {X 0,Y 307.585,Z 430.061,A -85,B 0,C 180,E1 14176.902,E2 14176.902} C_VEL
LIN {X 0,Y 300.065,Z 415.284,A -85,B 0,C 180,E1 14175.325,E2 14175.325} C_VEL
LIN {X 0,Y 293.162,Z 397.821,A -85,B 0,C 180,E1 14171.95,E2 14171.95} C_VEL
LIN {X 0,Y 290.412,Z 391.166,A -85,B 0,C 180,E1 14170.595,E2 14170.595} C_VEL
LIN {X 0,Y 290.337,Z 390.633,A -85,B 0,C 180,E1 14170.44,E2 14170.44} C_VEL
LIN {X 0,Y 290.307,Z 390.637,A -85,B 0,C 180,E1 14165.839,E2 14165.839} C_VEL
LIN {X 0,Y 290.299,Z 390.638,A -85,B 0,C 180,E1 14161.107,E2 14161.107} C_VEL
LIN {X 0,Y 290.313,Z 390.633,A -85,B 0,C 180,E1 14156.598,E2 14156.598} C_VEL
LIN {X 0,Y 290.328,Z 390.634,A -85,B 0,C 180,E1 14152.048,E2 14152.048} C_VEL
LIN {X 0,Y 290.3,Z 390.631,A -85,B 0,C 180,E1 14147.435,E2 14147.435} C_VEL
LIN {X 0,Y 290.299,Z 390.63,A -85,B 0,C 180,E1 14142.734,E2 14142.734} C_VEL
LIN {X 0,Y 290.328,Z 390.627,A -85,B 0,C 180,E1 14138.117,E2 14138.117} C_VEL
LIN {X 0,Y 290.304,Z 390.627,A -85,B 0,C 180,E1 14133.554,E2 14133.554} C_VEL
LIN {X 0,Y 290.293,Z 390.63,A -85,B 0,C 180,E1 14128.816,E2 14128.816} C_VEL
LIN {X 0,Y 290.321,Z 390.635,A -85,B 0,C 180,E1 14124.07,E2 14124.07} C_VEL
LIN {X 0,Y 290.309,Z 390.636,A -85,B 0,C 180,E1 14119.482,E2 14119.482} C_VEL
LIN {X 0,Y 290.292,Z 390.639,A -85,B 0,C 180,E1 14114.825,E2 14114.825} C_VEL
LIN {X 0,Y 290.304,Z 390.639,A -85,B 0,C 180,E1 14110.273,E2 14110.273} C_VEL
LIN {X 0,Y 290.32,Z 390.632,A -85,B 0,C 180,E1 14105.805,E2 14105.805} C_VEL
LIN {X 0,Y 290.306,Z 390.635,A -85,B 0,C 180,E1 14101.172,E2 14101.172} C_VEL
LIN {X 0,Y 290.294,Z 390.642,A -85,B 0,C 180,E1 14096.558,E2 14096.558} C_VEL
LIN {X 0,Y 290.308,Z 390.64,A -85,B 0,C 180,E1 14091.939,E2 14091.939} C_VEL
LIN {X 0,Y 290.322,Z 390.635,A -85,B 0,C 180,E1 14087.478,E2 14087.478} C_VEL
LIN {X 0,Y 290.32,Z 390.835,A -85,B 0,C 180,E1 14086.323,E2 14086.323} C_VEL
LIN {X 0,Y 295.072,Z 406.551,A -85,B 0,C 180,E1 14082.09,E2 14082.09} C_VEL
LIN {X 0,Y 299.706,Z 423.469,A -85,B 0,C 180,E1 14077.869,E2 14077.869} C_VEL
LIN {X 0,Y 303.844,Z 440.192,A -85,B 0,C 180,E1 14073.977,E2 14073.977} C_VEL
LIN {X 0,Y 303.298,Z 444.933,A -85,B 0,C 180,E1 14073.066,E2 14073.066} C_VEL
LIN {X 0,Y 301.345,Z 457.514,A -85,B 0,C 180,E1 14070.704,E2 14070.704} C_VEL
LIN {X 0,Y 299.816,Z 461.275,A -85,B 0,C 180,E1 14070.076,E2 14070.076} C_VEL
LIN {X 0,Y 292.503,Z 471.303,A -85,B 0,C 180,E1 14068.637,E2 14068.637} C_VEL
LIN {X 0,Y 291.309,Z 474.549,A -85,B 0,C 180,E1 14068.072,E2 14068.072} C_VEL
LIN {X 0,Y 291.025,Z 477.256,A -85,B 0,C 180,E1 14067.63,E2 14067.63} C_VEL
LIN {X 0,Y 294.801,Z 517.075,A -85,B 0,C 180,E1 14065.717,E2 14065.717} C_VEL
LIN {X 0,Y 289.785,Z 612.184,A -85,B 0,C 180,E1 14062.085,E2 14062.085} C_VEL
LIN {X 0,Y 288.855,Z 629.841,A -85,B 0,C 180,E1 14061.047,E2 14061.047} C_VEL
LIN {X 0,Y 287.722,Z 646.521,A -85,B 0,C 180,E1 14059.7,E2 14059.7} C_VEL
LIN {X 0,Y 286.428,Z 662.603,A -85,B 0,C 180,E1 14057.995,E2 14057.995} C_VEL
LIN {X 0,Y 285.152,Z 678.183,A -85,B 0,C 180,E1 14055.873,E2 14055.873} C_VEL
LIN {X 0,Y 283.972,Z 692.279,A -85,B 0,C 180,E1 14053.438,E2 14053.438} C_VEL
LIN {X 0,Y 283.063,Z 704.396,A -85,B 0,C 180,E1 14050.79,E2 14050.79} C_VEL
LIN {X 0,Y 282.494,Z 713.991,A -85,B 0,C 180,E1 14048.139,E2 14048.139} C_VEL
LIN {X 0,Y 282.235,Z 721.685,A -85,B 0,C 180,E1 14045.443,E2 14045.443} C_VEL
LIN {X 0,Y 282.296,Z 728.083,A -85,B 0,C 180,E1 14042.436,E2 14042.436} C_VEL
LIN {X 0,Y 282.683,Z 732.331,A -85,B 0,C 180,E1 14039.595,E2 14039.595} C_VEL
LIN {X 0,Y 283.494,Z 735.01,A -85,B 0,C 180,E1 14036.563,E2 14036.563} C_VEL
LIN {X 0,Y 284.678,Z 735.868,A -85,B 0,C 180,E1 14033.75,E2 14033.75} C_VEL
LIN {X 0,Y 286.446,Z 734.95,A -85,B 0,C 180,E1 14030.76,E2 14030.76} C_VEL
LIN {X 0,Y 288.78,Z 732.264,A -85,B 0,C 180,E1 14027.807,E2 14027.807} C_VEL
LIN {X 0,Y 291.924,Z 727.27,A -85,B 0,C 180,E1 14024.709,E2 14024.709} C_VEL
LIN {X 0,Y 295.262,Z 721.039,A -85,B 0,C 180,E1 14022.052,E2 14022.052} C_VEL
LIN {X 0,Y 299.148,Z 712.862,A -85,B 0,C 180,E1 14019.455,E2 14019.455} C_VEL
LIN {X 0,Y 303.28,Z 703.375,A -85,B 0,C 180,E1 14017.106,E2 14017.106} C_VEL
LIN {X 0,Y 308.268,Z 690.649,A -85,B 0,C 180,E1 14014.651,E2 14014.651} C_VEL
LIN {X 0,Y 313.495,Z 675.93,A -85,B 0,C 180,E1 14012.454,E2 14012.454} C_VEL
LIN {X 0,Y 318.595,Z 659.74,A -85,B 0,C 180,E1 14010.584,E2 14010.584} C_VEL
LIN {X 0,Y 323.415,Z 642.009,A -85,B 0,C 180,E1 14009.02,E2 14009.02} C_VEL
LIN {X 0,Y 327.538,Z 623.628,A -85,B 0,C 180,E1 14007.826,E2 14007.826} C_VEL
LIN {X 0,Y 341.562,Z 559.103,A -85,B 0,C 180,E1 14004.783,E2 14004.783} C_VEL
LIN {X 0,Y 346.184,Z 538.877,A -85,B 0,C 180,E1 14003.874,E2 14003.874} C_VEL
LIN {X 0,Y 348.373,Z 524.749,A -85,B 0,C 180,E1 14002.13,E2 14002.13} C_VEL
LIN {X 0,Y 350.82,Z 512.116,A -85,B 0,C 180,E1 14000.22,E2 14000.22} C_VEL
LIN {X 0,Y 351.421,Z 509.725,A -85,B 0,C 180,E1 13999.77,E2 13999.77} C_VEL
LIN {X 0,Y 351.958,Z 508.341,A -85,B 0,C 180,E1 13998.336,E2 13998.336} C_VEL
LIN {X 0,Y 352.815,Z 508.204,A -85,B 0,C 180,E1 13996.923,E2 13996.923} C_VEL
LIN {X 0,Y 352.966,Z 508.841,A -85,B 0,C 180,E1 13996.582,E2 13996.582} C_VEL
LIN {X 0,Y 351.915,Z 513.884,A -85,B 0,C 180,E1 13996.295,E2 13996.295} C_VEL
LIN {X 0,Y 337.737,Z 582.069,A -85,B 0,C 180,E1 13993.782,E2 13993.782} C_VEL
LIN {X 0,Y 325.623,Z 651.423,A -85,B 0,C 180,E1 13991.139,E2 13991.139} C_VEL
LIN {X 0,Y 321.129,Z 670.711,A -85,B 0,C 180,E1 13990.129,E2 13990.129} C_VEL
LIN {X 0,Y 315.616,Z 690.468,A -85,B 0,C 180,E1 13988.732,E2 13988.732} C_VEL
LIN {X 0,Y 310.101,Z 707.929,A -85,B 0,C 180,E1 13987.081,E2 13987.081} C_VEL
LIN {X 0,Y 304.477,Z 724.54,A -85,B 0,C 180,E1 13985.077,E2 13985.077} C_VEL
LIN {X 0,Y 299.135,Z 739.735,A -85,B 0,C 180,E1 13982.785,E2 13982.785} C_VEL
LIN {X 0,Y 294.23,Z 753.65,A -85,B 0,C 180,E1 13980.195,E2 13980.195} C_VEL
LIN {X 0,Y 289.629,Z 767.024,A -85,B 0,C 180,E1 13977.11,E2 13977.11} C_VEL
LIN {X 0,Y 285.729,Z 779.459,A -85,B 0,C 180,E1 13973.534,E2 13973.534} C_VEL
LIN {X 0,Y 283.581,Z 787.948,A -85,B 0,C 180,E1 13970.646,E2 13970.646} C_VEL
LIN {X 0,Y 281.976,Z 799.302,A -85,B 0,C 180,E1 13967.476,E2 13967.476} C_VEL
LIN {X 0,Y 280.979,Z 808.735,A -85,B 0,C 180,E1 13964.214,E2 13964.214} C_VEL
LIN {X 0,Y 280.464,Z 816.307,A -85,B 0,C 180,E1 13960.891,E2 13960.891} C_VEL
LIN {X 0,Y 280.388,Z 822.101,A -85,B 0,C 180,E1 13957.546,E2 13957.546} C_VEL
LIN {X 0,Y 280.482,Z 826.077,A -85,B 0,C 180,E1 13954.293,E2 13954.293} C_VEL
LIN {X 0,Y 280.554,Z 828.498,A -85,B 0,C 180,E1 13951.021,E2 13951.021} C_VEL
LIN {X 0,Y 280.431,Z 829.391,A -85,B 0,C 180,E1 13947.752,E2 13947.752} C_VEL
LIN {X 0,Y 280.232,Z 828.826,A -85,B 0,C 180,E1 13944.472,E2 13944.472} C_VEL
LIN {X 0,Y 280.212,Z 826.464,A -85,B 0,C 180,E1 13940.76,E2 13940.76} C_VEL
LIN {X 0,Y 280.755,Z 822.352,A -85,B 0,C 180,E1 13937.035,E2 13937.035} C_VEL
LIN {X 0,Y 282.212,Z 816.082,A -85,B 0,C 180,E1 13933.111,E2 13933.111} C_VEL
LIN {X 0,Y 284.606,Z 808.261,A -85,B 0,C 180,E1 13929.432,E2 13929.432} C_VEL
LIN {X 0,Y 288.101,Z 798.492,A -85,B 0,C 180,E1 13925.825,E2 13925.825} C_VEL
LIN {X 0,Y 292.763,Z 786.609,A -85,B 0,C 180,E1 13922.324,E2 13922.324} C_VEL
LIN {X 0,Y 298.307,Z 773.245,A -85,B 0,C 180,E1 13919.148,E2 13919.148} C_VEL
LIN {X 0,Y 304.581,Z 758.521,A -85,B 0,C 180,E1 13916.304,E2 13916.304} C_VEL
LIN {X 0,Y 311.698,Z 741.951,A -85,B 0,C 180,E1 13913.712,E2 13913.712} C_VEL
LIN {X 0,Y 319.318,Z 723.821,A -85,B 0,C 180,E1 13911.456,E2 13911.456} C_VEL
LIN {X 0,Y 327.041,Z 704.845,A -85,B 0,C 180,E1 13909.598,E2 13909.598} C_VEL
LIN {X 0,Y 334.664,Z 685.018,A -85,B 0,C 180,E1 13908.107,E2 13908.107} C_VEL
LIN {X 0,Y 341.896,Z 664.107,A -85,B 0,C 180,E1 13906.932,E2 13906.932} C_VEL
LIN {X 0,Y 349.29,Z 638.578,A -85,B 0,C 180,E1 13905.839,E2 13905.839} C_VEL
LIN {X 0,Y 357.714,Z 606,A -85,B 0,C 180,E1 13904.582,E2 13904.582} C_VEL
LIN {X 0,Y 347.698,Z 643.816,A -85,B 0,C 180,E1 13903.076,E2 13903.076} C_VEL
LIN {X 0,Y 341.975,Z 662.429,A -85,B 0,C 180,E1 13902.032,E2 13902.032} C_VEL
LIN {X 0,Y 335.339,Z 681.049,A -85,B 0,C 180,E1 13900.654,E2 13900.654} C_VEL
LIN {X 0,Y 328.069,Z 699.514,A -85,B 0,C 180,E1 13898.89,E2 13898.89} C_VEL
LIN {X 0,Y 320.642,Z 716.926,A -85,B 0,C 180,E1 13896.778,E2 13896.778} C_VEL
LIN {X 0,Y 313.496,Z 732.774,A -85,B 0,C 180,E1 13894.369,E2 13894.369} C_VEL
LIN {X 0,Y 306.749,Z 747.169,A -85,B 0,C 180,E1 13891.654,E2 13891.654} C_VEL
LIN {X 0,Y 300.495,Z 759.998,A -85,B 0,C 180,E1 13888.629,E2 13888.629} C_VEL
LIN {X 0,Y 294.89,Z 771.24,A -85,B 0,C 180,E1 13885.291,E2 13885.291} C_VEL
LIN {X 0,Y 290.311,Z 780.374,A -85,B 0,C 180,E1 13881.836,E2 13881.836} C_VEL
LIN {X 0,Y 286.71,Z 787.572,A -85,B 0,C 180,E1 13878.292,E2 13878.292} C_VEL
LIN {X 0,Y 283.917,Z 793.25,A -85,B 0,C 180,E1 13874.48,E2 13874.48} C_VEL
LIN {X 0,Y 282.049,Z 796.99,A -85,B 0,C 180,E1 13870.622,E2 13870.622} C_VEL
LIN {X 0,Y 280.989,Z 798.866,A -85,B 0,C 180,E1 13866.886,E2 13866.886} C_VEL
LIN {X 0,Y 280.469,Z 799.076,A -85,B 0,C 180,E1 13863.27,E2 13863.27} C_VEL
LIN {X 0,Y 280.282,Z 797.761,A -85,B 0,C 180,E1 13859.795,E2 13859.795} C_VEL
LIN {X 0,Y 280.245,Z 794.904,A -85,B 0,C 180,E1 13856.318,E2 13856.318} C_VEL
LIN {X 0,Y 280.425,Z 790.412,A -85,B 0,C 180,E1 13852.831,E2 13852.831} C_VEL
LIN {X 0,Y 280.917,Z 784.16,A -85,B 0,C 180,E1 13849.334,E2 13849.334} C_VEL
LIN {X 0,Y 281.845,Z 775.946,A -85,B 0,C 180,E1 13845.831,E2 13845.831} C_VEL
LIN {X 0,Y 283.225,Z 766.211,A -85,B 0,C 180,E1 13842.538,E2 13842.538} C_VEL
LIN {X 0,Y 285.172,Z 754.21,A -85,B 0,C 180,E1 13839.26,E2 13839.26} C_VEL
LIN {X 0,Y 287.498,Z 740.87,A -85,B 0,C 180,E1 13836.289,E2 13836.289} C_VEL
LIN {X 0,Y 290.101,Z 726.155,A -85,B 0,C 180,E1 13833.601,E2 13833.601} C_VEL
LIN {X 0,Y 292.831,Z 710.178,A -85,B 0,C 180,E1 13831.22,E2 13831.22} C_VEL
LIN {X 0,Y 295.669,Z 692.412,A -85,B 0,C 180,E1 13829.068,E2 13829.068} C_VEL
LIN {X 0,Y 298.353,Z 673.829,A -85,B 0,C 180,E1 13827.264,E2 13827.264} C_VEL
LIN {X 0,Y 300.717,Z 654.746,A -85,B 0,C 180,E1 13825.812,E2 13825.812} C_VEL
LIN {X 0,Y 302.731,Z 634.402,A -85,B 0,C 180,E1 13824.663,E2 13824.663} C_VEL
LIN {X 0,Y 304.384,Z 611.536,A -85,B 0,C 180,E1 13823.774,E2 13823.774} C_VEL
LIN {X 0,Y 314.694,Z 462.021,A -85,B 0,C 180,E1 13819.004,E2 13819.004} C_VEL
LIN {X 0,Y 300.564,Z 432.406,A -85,B 0,C 180,E1 13816.141,E2 13816.141} C_VEL
LIN {X 0,Y 292.051,Z 415.753,A -85,B 0,C 180,E1 13814.3,E2 13814.3} C_VEL
LIN {X 0,Y 284.86,Z 398.11,A -85,B 0,C 180,E1 13810.758,E2 13810.758} C_VEL
LIN {X 0,Y 282.356,Z 391.626,A -85,B 0,C 180,E1 13809.412,E2 13809.412} C_VEL
LIN {X 0,Y 282.37,Z 391.628,A -85,B 0,C 180,E1 13804.757,E2 13804.757} C_VEL
LIN {X 0,Y 282.392,Z 391.624,A -85,B 0,C 180,E1 13800.184,E2 13800.184} C_VEL
LIN {X 0,Y 282.364,Z 391.626,A -85,B 0,C 180,E1 13795.595,E2 13795.595} C_VEL
LIN {X 0,Y 282.366,Z 391.62,A -85,B 0,C 180,E1 13790.738,E2 13790.738} C_VEL
LIN {X 0,Y 282.385,Z 391.623,A -85,B 0,C 180,E1 13786.032,E2 13786.032} C_VEL
LIN {X 0,Y 282.361,Z 391.627,A -85,B 0,C 180,E1 13781.438,E2 13781.438} C_VEL
LIN {X 0,Y 282.36,Z 391.624,A -85,B 0,C 180,E1 13776.711,E2 13776.711} C_VEL
LIN {X 0,Y 282.38,Z 391.62,A -85,B 0,C 180,E1 13772.029,E2 13772.029} C_VEL
LIN {X 0,Y 282.369,Z 391.615,A -85,B 0,C 180,E1 13767.565,E2 13767.565} C_VEL
LIN {X 0,Y 282.352,Z 391.619,A -85,B 0,C 180,E1 13762.88,E2 13762.88} C_VEL
LIN {X 0,Y 282.371,Z 391.622,A -85,B 0,C 180,E1 13758.148,E2 13758.148} C_VEL
LIN {X 0,Y 282.377,Z 391.621,A -85,B 0,C 180,E1 13753.544,E2 13753.544} C_VEL
LIN {X 0,Y 282.356,Z 391.624,A -85,B 0,C 180,E1 13748.826,E2 13748.826} C_VEL
LIN {X 0,Y 282.369,Z 391.625,A -85,B 0,C 180,E1 13744.081,E2 13744.081} C_VEL
LIN {X 0,Y 282.393,Z 391.624,A -85,B 0,C 180,E1 13739.581,E2 13739.581} C_VEL
LIN {X 0,Y 282.358,Z 391.633,A -85,B 0,C 180,E1 13734.885,E2 13734.885} C_VEL
LIN {X 0,Y 282.36,Z 391.628,A -85,B 0,C 180,E1 13730.138,E2 13730.138} C_VEL
LIN {X 0,Y 282.384,Z 391.683,A -85,B 0,C 180,E1 13727.265,E2 13727.265} C_VEL
LIN {X 0,Y 287.406,Z 408.376,A -85,B 0,C 180,E1 13722.64,E2 13722.64} C_VEL
LIN {X 0,Y 291.836,Z 424.57,A -85,B 0,C 180,E1 13718.492,E2 13718.492} C_VEL
LIN {X 0,Y 295.988,Z 441.313,A -85,B 0,C 180,E1 13714.488,E2 13714.488} C_VEL
LIN {X 0,Y 296.165,Z 443.729,A -85,B 0,C 180,E1 13713.969,E2 13713.969} C_VEL
LIN {X 0,Y 291.945,Z 470.337,A -85,B 0,C 180,E1 13708.875,E2 13708.875} C_VEL
LIN {X 0,Y 291.309,Z 474.549,A -85,B 0,C 180,E1 13708.072,E2 13708.072} C_VEL
LIN {X 0,Y 290.229,Z 477.229,A -85,B 0,C 180,E1 13707.785,E2 13707.785} C_VEL
LIN {X 0,Y 286.227,Z 482.979,A -85,B 0,C 180,E1 13707.745,E2 13707.745} C_VEL
LIN {X 0,Y 283.157,Z 488.294,A -85,B 0,C 180,E1 13707.748,E2 13707.748} C_VEL
LIN {X 0,Y 282.245,Z 491.806,A -85,B 0,C 180,E1 13707.678,E2 13707.678} C_VEL
LIN {X 0,Y 282.659,Z 496.474,A -85,B 0,C 180,E1 13707.468,E2 13707.468} C_VEL
LIN {X 0,Y 286.244,Z 507.738,A -85,B 0,C 180,E1 13706.689,E2 13706.689} C_VEL
LIN {X 0,Y 286.42,Z 508.934,A -85,B 0,C 180,E1 13706.626,E2 13706.626} C_VEL
LIN {X 0,Y 287.168,Z 518.019,A -85,B 0,C 180,E1 13706.188,E2 13706.188} C_VEL
LIN {X 0,Y 282.007,Z 612.296,A -85,B 0,C 180,E1 13702.46,E2 13702.46} C_VEL
LIN {X 0,Y 281.039,Z 630.049,A -85,B 0,C 180,E1 13701.387,E2 13701.387} C_VEL
LIN {X 0,Y 279.827,Z 647.283,A -85,B 0,C 180,E1 13699.953,E2 13699.953} C_VEL
LIN {X 0,Y 278.499,Z 663.385,A -85,B 0,C 180,E1 13698.201,E2 13698.201} C_VEL
LIN {X 0,Y 277.192,Z 679.045,A -85,B 0,C 180,E1 13696.019,E2 13696.019} C_VEL
LIN {X 0,Y 275.988,Z 693.231,A -85,B 0,C 180,E1 13693.514,E2 13693.514} C_VEL
LIN {X 0,Y 275.094,Z 704.988,A -85,B 0,C 180,E1 13690.895,E2 13690.895} C_VEL
LIN {X 0,Y 274.512,Z 714.699,A -85,B 0,C 180,E1 13688.167,E2 13688.167} C_VEL
LIN {X 0,Y 274.251,Z 722.937,A -85,B 0,C 180,E1 13685.23,E2 13685.23} C_VEL
LIN {X 0,Y 274.362,Z 729.498,A -85,B 0,C 180,E1 13682.089,E2 13682.089} C_VEL
LIN {X 0,Y 274.832,Z 733.744,A -85,B 0,C 180,E1 13679.166,E2 13679.166} C_VEL
LIN {X 0,Y 275.749,Z 736.471,A -85,B 0,C 180,E1 13676.05,E2 13676.05} C_VEL
LIN {X 0,Y 277.196,Z 737.361,A -85,B 0,C 180,E1 13672.956,E2 13672.956} C_VEL
LIN {X 0,Y 279.356,Z 736.298,A -85,B 0,C 180,E1 13669.691,E2 13669.691} C_VEL
LIN {X 0,Y 282.014,Z 733.448,A -85,B 0,C 180,E1 13666.677,E2 13666.677} C_VEL
LIN {X 0,Y 285.559,Z 728.354,A -85,B 0,C 180,E1 13663.524,E2 13663.524} C_VEL
LIN {X 0,Y 289.26,Z 722.014,A -85,B 0,C 180,E1 13660.83,E2 13660.83} C_VEL
LIN {X 0,Y 293.568,Z 713.853,A -85,B 0,C 180,E1 13658.208,E2 13658.208} C_VEL
LIN {X 0,Y 298.814,Z 702.676,A -85,B 0,C 180,E1 13655.486,E2 13655.486} C_VEL
LIN {X 0,Y 304.141,Z 690.154,A -85,B 0,C 180,E1 13653.126,E2 13653.126} C_VEL
LIN {X 0,Y 309.421,Z 676.531,A -85,B 0,C 180,E1 13651.113,E2 13651.113} C_VEL
LIN {X 0,Y 314.697,Z 661.296,A -85,B 0,C 180,E1 13649.34,E2 13649.34} C_VEL
LIN {X 0,Y 319.861,Z 644.012,A -85,B 0,C 180,E1 13647.794,E2 13647.794} C_VEL
LIN {X 0,Y 324.359,Z 625.82,A -85,B 0,C 180,E1 13646.59,E2 13646.59} C_VEL
LIN {X 0,Y 337.598,Z 568.29,A -85,B 0,C 180,E1 13643.848,E2 13643.848} C_VEL
LIN {X 0,Y 344.028,Z 541.603,A -85,B 0,C 180,E1 13642.649,E2 13642.649} C_VEL
LIN {X 0,Y 346.732,Z 527.999,A -85,B 0,C 180,E1 13640.909,E2 13640.909} C_VEL
LIN {X 0,Y 349.493,Z 516.816,A -85,B 0,C 180,E1 13639.165,E2 13639.165} C_VEL
LIN {X 0,Y 350.28,Z 515.903,A -85,B 0,C 180,E1 13637.673,E2 13637.673} C_VEL
LIN {X 0,Y 350.319,Z 516.08,A -85,B 0,C 180,E1 13637.532,E2 13637.532} C_VEL
LIN {X 0,Y 334.98,Z 584.079,A -85,B 0,C 180,E1 13635.025,E2 13635.025} C_VEL
LIN {X 0,Y 322.189,Z 650.545,A -85,B 0,C 180,E1 13632.453,E2 13632.453} C_VEL
LIN {X 0,Y 316.964,Z 670.941,A -85,B 0,C 180,E1 13631.366,E2 13631.366} C_VEL
LIN {X 0,Y 311.157,Z 689.965,A -85,B 0,C 180,E1 13629.992,E2 13629.992} C_VEL
LIN {X 0,Y 305.289,Z 706.998,A -85,B 0,C 180,E1 13628.363,E2 13628.363} C_VEL
LIN {X 0,Y 299.363,Z 723.095,A -85,B 0,C 180,E1 13626.397,E2 13626.397} C_VEL
LIN {X 0,Y 293.532,Z 738.269,A -85,B 0,C 180,E1 13624.079,E2 13624.079} C_VEL
LIN {X 0,Y 288.006,Z 752.452,A -85,B 0,C 180,E1 13621.383,E2 13621.383} C_VEL
LIN {X 0,Y 282.969,Z 765.649,A -85,B 0,C 180,E1 13618.261,E2 13618.261} C_VEL
LIN {X 0,Y 278.826,Z 777.413,A -85,B 0,C 180,E1 13614.807,E2 13614.807} C_VEL
LIN {X 0,Y 275.764,Z 787.693,A -85,B 0,C 180,E1 13611.036,E2 13611.036} C_VEL
LIN {X 0,Y 275.26,Z 790.007,A -85,B 0,C 180,E1 13610.187,E2 13610.187} C_VEL
LIN {X 0,Y 273.737,Z 801.055,A -85,B 0,C 180,E1 13606.866,E2 13606.866} C_VEL
LIN {X 0,Y 272.852,Z 809.897,A -85,B 0,C 180,E1 13603.564,E2 13603.564} C_VEL
LIN {X 0,Y 272.442,Z 817.093,A -85,B 0,C 180,E1 13600.146,E2 13600.146} C_VEL
LIN {X 0,Y 272.443,Z 822.49,A -85,B 0,C 180,E1 13596.744,E2 13596.744} C_VEL
LIN {X 0,Y 272.54,Z 826.201,A -85,B 0,C 180,E1 13593.365,E2 13593.365} C_VEL
LIN {X 0,Y 272.574,Z 828.268,A -85,B 0,C 180,E1 13590,E2 13590} C_VEL
LIN {X 0,Y 272.376,Z 828.808,A -85,B 0,C 180,E1 13586.633,E2 13586.633} C_VEL
LIN {X 0,Y 272.198,Z 827.807,A -85,B 0,C 180,E1 13583.038,E2 13583.038} C_VEL
LIN {X 0,Y 272.376,Z 824.841,A -85,B 0,C 180,E1 13578.995,E2 13578.995} C_VEL
LIN {X 0,Y 273.396,Z 819.958,A -85,B 0,C 180,E1 13574.95,E2 13574.95} C_VEL
LIN {X 0,Y 275.47,Z 813.139,A -85,B 0,C 180,E1 13570.933,E2 13570.933} C_VEL
LIN {X 0,Y 278.583,Z 804.806,A -85,B 0,C 180,E1 13567.193,E2 13567.193} C_VEL
LIN {X 0,Y 282.874,Z 794.559,A -85,B 0,C 180,E1 13563.553,E2 13563.553} C_VEL
LIN {X 0,Y 288.421,Z 782.237,A -85,B 0,C 180,E1 13560.053,E2 13560.053} C_VEL
LIN {X 0,Y 294.984,Z 768.144,A -85,B 0,C 180,E1 13556.847,E2 13556.847} C_VEL
LIN {X 0,Y 302.469,Z 752.337,A -85,B 0,C 180,E1 13553.956,E2 13553.956} C_VEL
LIN {X 0,Y 310.815,Z 734.729,A -85,B 0,C 180,E1 13551.385,E2 13551.385} C_VEL
LIN {X 0,Y 319.098,Z 716.862,A -85,B 0,C 180,E1 13549.326,E2 13549.326} C_VEL
LIN {X 0,Y 327.328,Z 698.201,A -85,B 0,C 180,E1 13547.659,E2 13547.659} C_VEL
LIN {X 0,Y 335.301,Z 678.762,A -85,B 0,C 180,E1 13546.344,E2 13546.344} C_VEL
LIN {X 0,Y 343.068,Z 657.42,A -85,B 0,C 180,E1 13545.263,E2 13545.263} C_VEL
LIN {X 0,Y 348.211,Z 640.829,A -85,B 0,C 180,E1 13544.571,E2 13544.571} C_VEL
LIN {X 0,Y 341.784,Z 660.618,A -85,B 0,C 180,E1 13543.546,E2 13543.546} C_VEL
LIN {X 0,Y 334.66,Z 679.275,A -85,B 0,C 180,E1 13542.239,E2 13542.239} C_VEL
LIN {X 0,Y 326.744,Z 697.611,A -85,B 0,C 180,E1 13540.561,E2 13540.561} C_VEL
LIN {X 0,Y 318.376,Z 715.595,A -85,B 0,C 180,E1 13538.449,E2 13538.449} C_VEL
LIN {X 0,Y 310.298,Z 731.841,A -85,B 0,C 180,E1 13536.022,E2 13536.022} C_VEL
LIN {X 0,Y 302.651,Z 746.585,A -85,B 0,C 180,E1 13533.258,E2 13533.258} C_VEL
LIN {X 0,Y 295.767,Z 759.458,A -85,B 0,C 180,E1 13530.245,E2 13530.245} C_VEL
LIN {X 0,Y 289.519,Z 770.763,A -85,B 0,C 180,E1 13526.898,E2 13526.898} C_VEL
LIN {X 0,Y 284.29,Z 780.095,A -85,B 0,C 180,E1 13523.371,E2 13523.371} C_VEL
LIN {X 0,Y 280.007,Z 787.707,A -85,B 0,C 180,E1 13519.612,E2 13519.612} C_VEL
LIN {X 0,Y 276.777,Z 793.459,A -85,B 0,C 180,E1 13515.72,E2 13515.72} C_VEL
LIN {X 0,Y 274.562,Z 797.352,A -85,B 0,C 180,E1 13511.767,E2 13511.767} C_VEL
LIN {X 0,Y 273.218,Z 799.422,A -85,B 0,C 180,E1 13507.782,E2 13507.782} C_VEL
LIN {X 0,Y 272.562,Z 799.705,A -85,B 0,C 180,E1 13503.996,E2 13503.996} C_VEL
LIN {X 0,Y 272.295,Z 798.324,A -85,B 0,C 180,E1 13500.21,E2 13500.21} C_VEL
LIN {X 0,Y 272.245,Z 795.455,A -85,B 0,C 180,E1 13496.631,E2 13496.631} C_VEL
LIN {X 0,Y 272.406,Z 790.957,A -85,B 0,C 180,E1 13493.043,E2 13493.043} C_VEL
LIN {X 0,Y 272.891,Z 784.698,A -85,B 0,C 180,E1 13489.444,E2 13489.444} C_VEL
LIN {X 0,Y 273.826,Z 776.474,A -85,B 0,C 180,E1 13485.839,E2 13485.839} C_VEL
LIN {X 0,Y 275.229,Z 766.73,A -85,B 0,C 180,E1 13482.45,E2 13482.45} C_VEL
LIN {X 0,Y 277.221,Z 754.717,A -85,B 0,C 180,E1 13479.08,E2 13479.08} C_VEL
LIN {X 0,Y 279.588,Z 741.482,A -85,B 0,C 180,E1 13476.052,E2 13476.052} C_VEL
LIN {X 0,Y 282.284,Z 726.629,A -85,B 0,C 180,E1 13473.266,E2 13473.266} C_VEL
LIN {X 0,Y 285.093,Z 710.651,A -85,B 0,C 180,E1 13470.824,E2 13470.824} C_VEL
LIN {X 0,Y 288.012,Z 692.903,A -85,B 0,C 180,E1 13468.618,E2 13468.618} C_VEL
LIN {X 0,Y 290.764,Z 674.438,A -85,B 0,C 180,E1 13466.777,E2 13466.777} C_VEL
LIN {X 0,Y 293.26,Z 654.93,A -85,B 0,C 180,E1 13465.254,E2 13465.254} C_VEL
LIN {X 0,Y 295.351,Z 634.477,A -85,B 0,C 180,E1 13464.072,E2 13464.072} C_VEL
LIN {X 0,Y 297.104,Z 611.045,A -85,B 0,C 180,E1 13463.139,E2 13463.139} C_VEL
LIN {X 0,Y 307.624,Z 464.337,A -85,B 0,C 180,E1 13458.31,E2 13458.31} C_VEL
LIN {X 0,Y 294.283,Z 436.284,A -85,B 0,C 180,E1 13455.521,E2 13455.521} C_VEL
LIN {X 0,Y 283.805,Z 415.69,A -85,B 0,C 180,E1 13453.116,E2 13453.116} C_VEL
LIN {X 0,Y 277.021,Z 399.25,A -85,B 0,C 180,E1 13449.707,E2 13449.707} C_VEL
LIN {X 0,Y 274.485,Z 392.852,A -85,B 0,C 180,E1 13448.343,E2 13448.343} C_VEL
LIN {X 0,Y 274.431,Z 392.615,A -85,B 0,C 180,E1 13443.829,E2 13443.829} C_VEL
LIN {X 0,Y 274.421,Z 392.613,A -85,B 0,C 180,E1 13438.986,E2 13438.986} C_VEL
LIN {X 0,Y 274.445,Z 392.609,A -85,B 0,C 180,E1 13434.311,E2 13434.311} C_VEL
LIN {X 0,Y 274.427,Z 392.616,A -85,B 0,C 180,E1 13429.585,E2 13429.585} C_VEL
LIN {X 0,Y 274.421,Z 392.617,A -85,B 0,C 180,E1 13424.776,E2 13424.776} C_VEL
LIN {X 0,Y 274.442,Z 392.611,A -85,B 0,C 180,E1 13420.071,E2 13420.071} C_VEL
LIN {X 0,Y 274.423,Z 392.611,A -85,B 0,C 180,E1 13415.436,E2 13415.436} C_VEL
LIN {X 0,Y 274.419,Z 392.614,A -85,B 0,C 180,E1 13410.626,E2 13410.626} C_VEL
LIN {X 0,Y 274.436,Z 392.611,A -85,B 0,C 180,E1 13405.821,E2 13405.821} C_VEL
LIN {X 0,Y 274.419,Z 392.612,A -85,B 0,C 180,E1 13401.197,E2 13401.197} C_VEL
LIN {X 0,Y 274.426,Z 392.612,A -85,B 0,C 180,E1 13396.301,E2 13396.301} C_VEL
LIN {X 0,Y 274.44,Z 392.617,A -85,B 0,C 180,E1 13391.52,E2 13391.52} C_VEL
LIN {X 0,Y 274.417,Z 392.614,A -85,B 0,C 180,E1 13386.662,E2 13386.662} C_VEL
LIN {X 0,Y 274.446,Z 392.613,A -85,B 0,C 180,E1 13381.843,E2 13381.843} C_VEL
LIN {X 0,Y 274.426,Z 392.621,A -85,B 0,C 180,E1 13377.12,E2 13377.12} C_VEL
LIN {X 0,Y 274.418,Z 392.621,A -85,B 0,C 180,E1 13372.247,E2 13372.247} C_VEL
LIN {X 0,Y 274.448,Z 392.807,A -85,B 0,C 180,E1 13368.187,E2 13368.187} C_VEL
LIN {X 0,Y 278.961,Z 407.659,A -85,B 0,C 180,E1 13363.91,E2 13363.91} C_VEL
LIN {X 0,Y 283.401,Z 423.481,A -85,B 0,C 180,E1 13359.686,E2 13359.686} C_VEL
LIN {X 0,Y 287.437,Z 439.555,A -85,B 0,C 180,E1 13355.701,E2 13355.701} C_VEL
LIN {X 0,Y 288.57,Z 445.148,A -85,B 0,C 180,E1 13354.387,E2 13354.387} C_VEL
LIN {X 0,Y 284.17,Z 471.85,A -85,B 0,C 180,E1 13349.165,E2 13349.165} C_VEL
LIN {X 0,Y 283.45,Z 477.104,A -85,B 0,C 180,E1 13348.209,E2 13348.209} C_VEL
LIN {X 0,Y 286.42,Z 508.934,A -85,B 0,C 180,E1 13346.626,E2 13346.626} C_VEL
LIN {X 0,Y 286.136,Z 515.42,A -85,B 0,C 180,E1 13346.372,E2 13346.372} C_VEL
LIN {X 0,Y 283.328,Z 525.012,A -85,B 0,C 180,E1 13346.153,E2 13346.153} C_VEL
LIN {X 0,Y 278.868,Z 537.817,A -85,B 0,C 180,E1 13345.888,E2 13345.888} C_VEL
LIN {X 0,Y 277.987,Z 543.315,A -85,B 0,C 180,E1 13345.701,E2 13345.701} C_VEL
LIN {X 0,Y 274.148,Z 613.698,A -85,B 0,C 180,E1 13342.765,E2 13342.765} C_VEL
LIN {X 0,Y 273.124,Z 631.677,A -85,B 0,C 180,E1 13341.625,E2 13341.625} C_VEL
LIN {X 0,Y 271.89,Z 648.549,A -85,B 0,C 180,E1 13340.165,E2 13340.165} C_VEL
LIN {X 0,Y 270.5,Z 664.979,A -85,B 0,C 180,E1 13338.312,E2 13338.312} C_VEL
LIN {X 0,Y 269.233,Z 679.887,A -85,B 0,C 180,E1 13336.173,E2 13336.173} C_VEL
LIN {X 0,Y 267.998,Z 694.066,A -85,B 0,C 180,E1 13333.594,E2 13333.594} C_VEL
LIN {X 0,Y 267.062,Z 706.297,A -85,B 0,C 180,E1 13330.789,E2 13330.789} C_VEL
LIN {X 0,Y 266.497,Z 716.034,A -85,B 0,C 180,E1 13327.98,E2 13327.98} C_VEL
LIN {X 0,Y 266.273,Z 723.792,A -85,B 0,C 180,E1 13325.171,E2 13325.171} C_VEL
LIN {X 0,Y 266.407,Z 730.462,A -85,B 0,C 180,E1 13321.936,E2 13321.936} C_VEL
LIN {X 0,Y 266.933,Z 734.917,A -85,B 0,C 180,E1 13318.927,E2 13318.927} C_VEL
LIN {X 0,Y 267.94,Z 737.788,A -85,B 0,C 180,E1 13315.72,E2 13315.72} C_VEL
LIN {X 0,Y 269.526,Z 738.898,A -85,B 0,C 180,E1 13312.54,E2 13312.54} C_VEL
LIN {X 0,Y 271.872,Z 738.04,A -85,B 0,C 180,E1 13309.19,E2 13309.19} C_VEL
LIN {X 0,Y 274.75,Z 735.443,A -85,B 0,C 180,E1 13306.103,E2 13306.103} C_VEL
LIN {X 0,Y 278.299,Z 730.999,A -85,B 0,C 180,E1 13303.082,E2 13303.082} C_VEL
LIN {X 0,Y 282.554,Z 724.699,A -85,B 0,C 180,E1 13300.141,E2 13300.141} C_VEL
LIN {X 0,Y 287.843,Z 715.625,A -85,B 0,C 180,E1 13297.105,E2 13297.105} C_VEL
LIN {X 0,Y 293.528,Z 704.715,A -85,B 0,C 180,E1 13294.367,E2 13294.367} C_VEL
LIN {X 0,Y 299.275,Z 692.55,A -85,B 0,C 180,E1 13292.005,E2 13292.005} C_VEL
LIN {X 0,Y 305.181,Z 678.792,A -85,B 0,C 180,E1 13289.916,E2 13289.916} C_VEL
LIN {X 0,Y 311.086,Z 663.293,A -85,B 0,C 180,E1 13288.081,E2 13288.081} C_VEL
LIN {X 0,Y 316.315,Z 647.485,A -85,B 0,C 180,E1 13286.633,E2 13286.633} C_VEL
LIN {X 0,Y 321.077,Z 630.408,A -85,B 0,C 180,E1 13285.448,E2 13285.448} C_VEL
LIN {X 0,Y 330.703,Z 590.468,A -85,B 0,C 180,E1 13283.471,E2 13283.471} C_VEL
LIN {X 0,Y 342.331,Z 544.605,A -85,B 0,C 180,E1 13281.422,E2 13281.422} C_VEL
LIN {X 0,Y 345.334,Z 532.159,A -85,B 0,C 180,E1 13279.785,E2 13279.785} C_VEL
LIN {X 0,Y 347.577,Z 524.523,A -85,B 0,C 180,E1 13278.564,E2 13278.564} C_VEL
LIN {X 0,Y 331.71,Z 590.439,A -85,B 0,C 180,E1 13276.135,E2 13276.135} C_VEL
LIN {X 0,Y 319.19,Z 649.844,A -85,B 0,C 180,E1 13273.811,E2 13273.811} C_VEL
LIN {X 0,Y 313.349,Z 670.698,A -85,B 0,C 180,E1 13272.693,E2 13272.693} C_VEL
LIN {X 0,Y 307.225,Z 689.081,A -85,B 0,C 180,E1 13271.351,E2 13271.351} C_VEL
LIN {X 0,Y 300.984,Z 705.749,A -85,B 0,C 180,E1 13269.753,E2 13269.753} C_VEL
LIN {X 0,Y 294.558,Z 721.775,A -85,B 0,C 180,E1 13267.785,E2 13267.785} C_VEL
LIN {X 0,Y 288.36,Z 736.55,A -85,B 0,C 180,E1 13265.506,E2 13265.506} C_VEL
LIN {X 0,Y 282.342,Z 750.582,A -85,B 0,C 180,E1 13262.808,E2 13262.808} C_VEL
LIN {X 0,Y 276.796,Z 763.681,A -85,B 0,C 180,E1 13259.662,E2 13259.662} C_VEL
LIN {X 0,Y 272.126,Z 775.407,A -85,B 0,C 180,E1 13256.162,E2 13256.162} C_VEL
LIN {X 0,Y 268.564,Z 785.692,A -85,B 0,C 180,E1 13252.318,E2 13252.318} C_VEL
LIN {X 0,Y 267.074,Z 791.065,A -85,B 0,C 180,E1 13249.919,E2 13249.919} C_VEL
LIN {X 0,Y 265.65,Z 801.476,A -85,B 0,C 180,E1 13246.622,E2 13246.622} C_VEL
LIN {X 0,Y 264.777,Z 810.565,A -85,B 0,C 180,E1 13243.027,E2 13243.027} C_VEL
LIN {X 0,Y 264.448,Z 817.817,A -85,B 0,C 180,E1 13239.313,E2 13239.313} C_VEL
LIN {X 0,Y 264.503,Z 822.781,A -85,B 0,C 180,E1 13235.858,E2 13235.858} C_VEL
LIN {X 0,Y 264.604,Z 826.145,A -85,B 0,C 180,E1 13232.382,E2 13232.382} C_VEL
LIN {X 0,Y 264.564,Z 827.88,A -85,B 0,C 180,E1 13229.134,E2 13229.134} C_VEL
LIN {X 0,Y 264.314,Z 828.198,A -85,B 0,C 180,E1 13225.444,E2 13225.444} C_VEL
LIN {X 0,Y 264.185,Z 826.883,A -85,B 0,C 180,E1 13221.731,E2 13221.731} C_VEL
LIN {X 0,Y 264.574,Z 823.839,A -85,B 0,C 180,E1 13217.782,E2 13217.782} C_VEL
LIN {X 0,Y 265.938,Z 818.811,A -85,B 0,C 180,E1 13213.621,E2 13213.621} C_VEL
LIN {X 0,Y 268.472,Z 811.877,A -85,B 0,C 180,E1 13209.508,E2 13209.508} C_VEL
LIN {X 0,Y 272.339,Z 802.989,A -85,B 0,C 180,E1 13205.489,E2 13205.489} C_VEL
LIN {X 0,Y 277.591,Z 791.974,A -85,B 0,C 180,E1 13201.611,E2 13201.611} C_VEL
LIN {X 0,Y 284.169,Z 778.998,A -85,B 0,C 180,E1 13197.991,E2 13197.991} C_VEL
LIN {X 0,Y 292.057,Z 763.919,A -85,B 0,C 180,E1 13194.649,E2 13194.649} C_VEL
LIN {X 0,Y 300.656,Z 747.682,A -85,B 0,C 180,E1 13191.789,E2 13191.789} C_VEL
LIN {X 0,Y 309.612,Z 730.495,A -85,B 0,C 180,E1 13189.404,E2 13189.404} C_VEL
LIN {X 0,Y 319.027,Z 711.928,A -85,B 0,C 180,E1 13187.393,E2 13187.393} C_VEL
LIN {X 0,Y 328.015,Z 693.193,A -85,B 0,C 180,E1 13185.851,E2 13185.851} C_VEL
LIN {X 0,Y 336.617,Z 673.584,A -85,B 0,C 180,E1 13184.652,E2 13184.652} C_VEL
LIN {X 0,Y 338.319,Z 669.346,A -85,B 0,C 180,E1 13184.418,E2 13184.418} C_VEL
LIN {X 0,Y 330.357,Z 687.438,A -85,B 0,C 180,E1 13183.039,E2 13183.039} C_VEL
LIN {X 0,Y 321.824,Z 704.793,A -85,B 0,C 180,E1 13181.315,E2 13181.315} C_VEL
LIN {X 0,Y 312.525,Z 722.388,A -85,B 0,C 180,E1 13179.069,E2 13179.069} C_VEL
LIN {X 0,Y 303.887,Z 737.882,A -85,B 0,C 180,E1 13176.55,E2 13176.55} C_VEL
LIN {X 0,Y 295.715,Z 751.884,A -85,B 0,C 180,E1 13173.677,E2 13173.677} C_VEL
LIN {X 0,Y 288.181,Z 764.422,A -85,B 0,C 180,E1 13170.434,E2 13170.434} C_VEL
LIN {X 0,Y 281.77,Z 774.864,A -85,B 0,C 180,E1 13167.014,E2 13167.014} C_VEL
LIN {X 0,Y 276.186,Z 783.733,A -85,B 0,C 180,E1 13163.241,E2 13163.241} C_VEL
LIN {X 0,Y 271.799,Z 790.62,A -85,B 0,C 180,E1 13159.334,E2 13159.334} C_VEL
LIN {X 0,Y 268.423,Z 795.852,A -85,B 0,C 180,E1 13155.114,E2 13155.114} C_VEL
LIN {X 0,Y 266.292,Z 798.971,A -85,B 0,C 180,E1 13151.04,E2 13151.04} C_VEL
LIN {X 0,Y 265.094,Z 800.276,A -85,B 0,C 180,E1 13147.15,E2 13147.15} C_VEL
LIN {X 0,Y 264.489,Z 799.969,A -85,B 0,C 180,E1 13143.25,E2 13143.25} C_VEL
LIN {X 0,Y 264.284,Z 798.15,A -85,B 0,C 180,E1 13139.566,E2 13139.566} C_VEL
LIN {X 0,Y 264.258,Z 794.79,A -85,B 0,C 180,E1 13135.877,E2 13135.877} C_VEL
LIN {X 0,Y 264.503,Z 789.584,A -85,B 0,C 180,E1 13132.056,E2 13132.056} C_VEL
LIN {X 0,Y 265.08,Z 782.955,A -85,B 0,C 180,E1 13128.468,E2 13128.468} C_VEL
LIN {X 0,Y 266.12,Z 774.587,A -85,B 0,C 180,E1 13124.928,E2 13124.928} C_VEL
LIN {X 0,Y 267.684,Z 764.44,A -85,B 0,C 180,E1 13121.488,E2 13121.488} C_VEL
LIN {X 0,Y 269.73,Z 752.654,A -85,B 0,C 180,E1 13118.242,E2 13118.242} C_VEL
LIN {X 0,Y 272.177,Z 739.329,A -85,B 0,C 180,E1 13115.242,E2 13115.242} C_VEL
LIN {X 0,Y 274.925,Z 724.487,A -85,B 0,C 180,E1 13112.491,E2 13112.491} C_VEL
LIN {X 0,Y 277.882,Z 708.021,A -85,B 0,C 180,E1 13109.99,E2 13109.99} C_VEL
LIN {X 0,Y 280.81,Z 690.591,A -85,B 0,C 180,E1 13107.838,E2 13107.838} C_VEL
LIN {X 0,Y 283.622,Z 671.952,A -85,B 0,C 180,E1 13105.999,E2 13105.999} C_VEL
LIN {X 0,Y 286.127,Z 652.195,A -85,B 0,C 180,E1 13104.488,E2 13104.488} C_VEL
LIN {X 0,Y 288.252,Z 631.468,A -85,B 0,C 180,E1 13103.312,E2 13103.312} C_VEL
LIN {X 0,Y 290.142,Z 605.875,A -85,B 0,C 180,E1 13102.327,E2 13102.327} C_VEL
LIN {X 0,Y 300.654,Z 466.815,A -85,B 0,C 180,E1 13097.609,E2 13097.609} C_VEL
LIN {X 0,Y 287.904,Z 439.98,A -85,B 0,C 180,E1 13094.865,E2 13094.865} C_VEL
LIN {X 0,Y 275.934,Z 416.658,A -85,B 0,C 180,E1 13092.095,E2 13092.095} C_VEL
LIN {X 0,Y 269.193,Z 400.415,A -85,B 0,C 180,E1 13088.609,E2 13088.609} C_VEL
LIN {X 0,Y 266.485,Z 393.606,A -85,B 0,C 180,E1 13087.089,E2 13087.089} C_VEL
LIN {X 0,Y 266.508,Z 393.601,A -85,B 0,C 180,E1 13082.191,E2 13082.191} C_VEL
LIN {X 0,Y 266.484,Z 393.603,A -85,B 0,C 180,E1 13077.484,E2 13077.484} C_VEL
LIN {X 0,Y 266.5,Z 393.601,A -85,B 0,C 180,E1 13072.5,E2 13072.5} C_VEL
LIN {X 0,Y 266.492,Z 393.598,A -85,B 0,C 180,E1 13067.692,E2 13067.692} C_VEL
LIN {X 0,Y 266.484,Z 393.597,A -85,B 0,C 180,E1 13062.699,E2 13062.699} C_VEL
LIN {X 0,Y 266.507,Z 393.595,A -85,B 0,C 180,E1 13057.921,E2 13057.921} C_VEL
LIN {X 0,Y 266.477,Z 393.596,A -85,B 0,C 180,E1 13053.011,E2 13053.011} C_VEL
LIN {X 0,Y 266.492,Z 393.591,A -85,B 0,C 180,E1 13048.28,E2 13048.28} C_VEL
LIN {X 0,Y 266.492,Z 393.597,A -85,B 0,C 180,E1 13043.537,E2 13043.537} C_VEL
LIN {X 0,Y 266.478,Z 393.602,A -85,B 0,C 180,E1 13038.749,E2 13038.749} C_VEL
LIN {X 0,Y 266.494,Z 393.604,A -85,B 0,C 180,E1 13034.104,E2 13034.104} C_VEL
LIN {X 0,Y 266.492,Z 393.6,A -85,B 0,C 180,E1 13029.348,E2 13029.348} C_VEL
LIN {X 0,Y 266.48,Z 393.603,A -85,B 0,C 180,E1 13024.438,E2 13024.438} C_VEL
LIN {X 0,Y 266.513,Z 393.602,A -85,B 0,C 180,E1 13019.571,E2 13019.571} C_VEL
LIN {X 0,Y 266.477,Z 393.611,A -85,B 0,C 180,E1 13014.702,E2 13014.702} C_VEL
LIN {X 0,Y 266.497,Z 393.604,A -85,B 0,C 180,E1 13009.81,E2 13009.81} C_VEL
LIN {X 0,Y 266.52,Z 393.777,A -85,B 0,C 180,E1 13009.178,E2 13009.178} C_VEL
LIN {X 0,Y 271.18,Z 409.04,A -85,B 0,C 180,E1 13004.634,E2 13004.634} C_VEL
LIN {X 0,Y 275.33,Z 423.897,A -85,B 0,C 180,E1 13000.545,E2 13000.545} C_VEL
LIN {X 0,Y 279.464,Z 440.125,A -85,B 0,C 180,E1 12996.389,E2 12996.389} C_VEL
LIN {X 0,Y 280.877,Z 447.048,A -85,B 0,C 180,E1 12994.72,E2 12994.72} C_VEL
LIN {X 0,Y 276.397,Z 473.318,A -85,B 0,C 180,E1 12989.471,E2 12989.471} C_VEL
LIN {X 0,Y 275.898,Z 477.002,A -85,B 0,C 180,E1 12988.808,E2 12988.808} C_VEL
LIN {X 0,Y 279.556,Z 518.61,A -85,B 0,C 180,E1 12986.685,E2 12986.685} C_VEL
LIN {X 0,Y 277.987,Z 543.315,A -85,B 0,C 180,E1 12985.701,E2 12985.701} C_VEL
LIN {X 0,Y 276.551,Z 550.858,A -85,B 0,C 180,E1 12985.459,E2 12985.459} C_VEL
LIN {X 0,Y 269.337,Z 570.728,A -85,B 0,C 180,E1 12985.005,E2 12985.005} C_VEL
LIN {X 0,Y 268.259,Z 577.208,A -85,B 0,C 180,E1 12984.776,E2 12984.776} C_VEL
LIN {X 0,Y 266.227,Z 616.388,A -85,B 0,C 180,E1 12983.016,E2 12983.016} C_VEL
LIN {X 0,Y 265.175,Z 633.856,A -85,B 0,C 180,E1 12981.833,E2 12981.833} C_VEL
LIN {X 0,Y 263.87,Z 650.678,A -85,B 0,C 180,E1 12980.287,E2 12980.287} C_VEL
LIN {X 0,Y 262.502,Z 666.361,A -85,B 0,C 180,E1 12978.43,E2 12978.43} C_VEL
LIN {X 0,Y 261.209,Z 681.148,A -85,B 0,C 180,E1 12976.227,E2 12976.227} C_VEL
LIN {X 0,Y 259.964,Z 695.344,A -85,B 0,C 180,E1 12973.569,E2 12973.569} C_VEL
LIN {X 0,Y 259.028,Z 707.613,A -85,B 0,C 180,E1 12970.678,E2 12970.678} C_VEL
LIN {X 0,Y 258.48,Z 717.324,A -85,B 0,C 180,E1 12967.781,E2 12967.781} C_VEL
LIN {X 0,Y 258.286,Z 725.573,A -85,B 0,C 180,E1 12964.663,E2 12964.663} C_VEL
LIN {X 0,Y 258.513,Z 732.21,A -85,B 0,C 180,E1 12961.33,E2 12961.33} C_VEL
LIN {X 0,Y 259.142,Z 736.539,A -85,B 0,C 180,E1 12958.231,E2 12958.231} C_VEL
LIN {X 0,Y 260.445,Z 739.528,A -85,B 0,C 180,E1 12954.714,E2 12954.714} C_VEL
LIN {X 0,Y 262.277,Z 740.437,A -85,B 0,C 180,E1 12951.45,E2 12951.45} C_VEL
LIN {X 0,Y 264.985,Z 739.479,A -85,B 0,C 180,E1 12948.023,E2 12948.023} C_VEL
LIN {X 0,Y 268.232,Z 736.778,A -85,B 0,C 180,E1 12944.875,E2 12944.875} C_VEL
LIN {X 0,Y 272.487,Z 731.944,A -85,B 0,C 180,E1 12941.605,E2 12941.605} C_VEL
LIN {X 0,Y 277.212,Z 725.431,A -85,B 0,C 180,E1 12938.636,E2 12938.636} C_VEL
LIN {X 0,Y 282.692,Z 716.958,A -85,B 0,C 180,E1 12935.778,E2 12935.778} C_VEL
LIN {X 0,Y 289.32,Z 705.393,A -85,B 0,C 180,E1 12932.86,E2 12932.86} C_VEL
LIN {X 0,Y 295.828,Z 692.734,A -85,B 0,C 180,E1 12930.432,E2 12930.432} C_VEL
LIN {X 0,Y 301.974,Z 679.554,A -85,B 0,C 180,E1 12928.456,E2 12928.456} C_VEL
LIN {X 0,Y 308.346,Z 664.287,A -85,B 0,C 180,E1 12926.659,E2 12926.659} C_VEL
LIN {X 0,Y 313.934,Z 648.675,A -85,B 0,C 180,E1 12925.243,E2 12925.243} C_VEL
LIN {X 0,Y 318.924,Z 632.232,A -85,B 0,C 180,E1 12924.108,E2 12924.108} C_VEL
LIN {X 0,Y 328.778,Z 593.711,A -85,B 0,C 180,E1 12922.209,E2 12922.209} C_VEL
LIN {X 0,Y 341.093,Z 547.702,A -85,B 0,C 180,E1 12920.176,E2 12920.176} C_VEL
LIN {X 0,Y 342.824,Z 541.329,A -85,B 0,C 180,E1 12919.324,E2 12919.324} C_VEL
LIN {X 0,Y 325.566,Z 610.464,A -85,B 0,C 180,E1 12916.756,E2 12916.756} C_VEL
LIN {X 0,Y 316.829,Z 648.67,A -85,B 0,C 180,E1 12915.24,E2 12915.24} C_VEL
LIN {X 0,Y 310.681,Z 668.961,A -85,B 0,C 180,E1 12914.168,E2 12914.168} C_VEL
LIN {X 0,Y 304.529,Z 686.194,A -85,B 0,C 180,E1 12912.944,E2 12912.944} C_VEL
LIN {X 0,Y 297.854,Z 702.823,A -85,B 0,C 180,E1 12911.4,E2 12911.4} C_VEL
LIN {X 0,Y 290.692,Z 719.291,A -85,B 0,C 180,E1 12909.417,E2 12909.417} C_VEL
LIN {X 0,Y 283.437,Z 735.137,A -85,B 0,C 180,E1 12906.975,E2 12906.975} C_VEL
LIN {X 0,Y 276.574,Z 749.653,A -85,B 0,C 180,E1 12904.12,E2 12904.12} C_VEL
LIN {X 0,Y 270.487,Z 762.626,A -85,B 0,C 180,E1 12900.919,E2 12900.919} C_VEL
LIN {X 0,Y 265.356,Z 774.151,A -85,B 0,C 180,E1 12897.368,E2 12897.368} C_VEL
LIN {X 0,Y 261.349,Z 784.297,A -85,B 0,C 180,E1 12893.446,E2 12893.446} C_VEL
LIN {X 0,Y 258.776,Z 792.807,A -85,B 0,C 180,E1 12889.408,E2 12889.408} C_VEL
LIN {X 0,Y 257.399,Z 803.419,A -85,B 0,C 180,E1 12885.778,E2 12885.778} C_VEL
LIN {X 0,Y 256.665,Z 811.947,A -85,B 0,C 180,E1 12882.099,E2 12882.099} C_VEL
LIN {X 0,Y 256.472,Z 818.688,A -85,B 0,C 180,E1 12878.294,E2 12878.294} C_VEL
LIN {X 0,Y 256.577,Z 823.282,A -85,B 0,C 180,E1 12874.694,E2 12874.694} C_VEL
LIN {X 0,Y 256.658,Z 826.189,A -85,B 0,C 180,E1 12871.116,E2 12871.116} C_VEL
LIN {X 0,Y 256.505,Z 827.48,A -85,B 0,C 180,E1 12867.766,E2 12867.766} C_VEL
LIN {X 0,Y 256.239,Z 827.406,A -85,B 0,C 180,E1 12863.952,E2 12863.952} C_VEL
LIN {X 0,Y 256.276,Z 825.615,A -85,B 0,C 180,E1 12859.888,E2 12859.888} C_VEL
LIN {X 0,Y 257.146,Z 821.911,A -85,B 0,C 180,E1 12855.59,E2 12855.59} C_VEL
LIN {X 0,Y 259.149,Z 816.363,A -85,B 0,C 180,E1 12851.323,E2 12851.323} C_VEL
LIN {X 0,Y 262.487,Z 808.954,A -85,B 0,C 180,E1 12847.136,E2 12847.136} C_VEL
LIN {X 0,Y 267.532,Z 799.087,A -85,B 0,C 180,E1 12842.873,E2 12842.873} C_VEL
LIN {X 0,Y 273.849,Z 787.65,A -85,B 0,C 180,E1 12839.015,E2 12839.015} C_VEL
LIN {X 0,Y 281.309,Z 774.689,A -85,B 0,C 180,E1 12835.548,E2 12835.548} C_VEL
LIN {X 0,Y 289.991,Z 759.831,A -85,B 0,C 180,E1 12832.39,E2 12832.39} C_VEL
LIN {X 0,Y 299.55,Z 743.469,A -85,B 0,C 180,E1 12829.643,E2 12829.643} C_VEL
LIN {X 0,Y 309.757,Z 725.764,A -85,B 0,C 180,E1 12827.323,E2 12827.323} C_VEL
LIN {X 0,Y 319.678,Z 707.875,A -85,B 0,C 180,E1 12825.524,E2 12825.524} C_VEL
LIN {X 0,Y 328.344,Z 691.184,A -85,B 0,C 180,E1 12824.232,E2 12824.232} C_VEL
LIN {X 0,Y 318.628,Z 708.933,A -85,B 0,C 180,E1 12822.429,E2 12822.429} C_VEL
LIN {X 0,Y 309.127,Z 725.131,A -85,B 0,C 180,E1 12820.307,E2 12820.307} C_VEL
LIN {X 0,Y 299.158,Z 741.09,A -85,B 0,C 180,E1 12817.616,E2 12817.616} C_VEL
LIN {X 0,Y 290.2,Z 754.909,A -85,B 0,C 180,E1 12814.645,E2 12814.645} C_VEL
LIN {X 0,Y 282.027,Z 767.134,A -85,B 0,C 180,E1 12811.305,E2 12811.305} C_VEL
LIN {X 0,Y 274.998,Z 777.285,A -85,B 0,C 180,E1 12807.735,E2 12807.735} C_VEL
LIN {X 0,Y 268.794,Z 786.077,A -85,B 0,C 180,E1 12803.687,E2 12803.687} C_VEL
LIN {X 0,Y 264.182,Z 792.497,A -85,B 0,C 180,E1 12799.684,E2 12799.684} C_VEL
LIN {X 0,Y 260.771,Z 797.099,A -85,B 0,C 180,E1 12795.569,E2 12795.569} C_VEL
LIN {X 0,Y 258.468,Z 799.929,A -85,B 0,C 180,E1 12791.378,E2 12791.378} C_VEL
LIN {X 0,Y 257.116,Z 800.991,A -85,B 0,C 180,E1 12787.148,E2 12787.148} C_VEL
LIN {X 0,Y 256.487,Z 800.355,A -85,B 0,C 180,E1 12783.128,E2 12783.128} C_VEL
LIN {X 0,Y 256.269,Z 798.059,A -85,B 0,C 180,E1 12779.106,E2 12779.106} C_VEL
LIN {X 0,Y 256.275,Z 794.298,A -85,B 0,C 180,E1 12775.3,E2 12775.3} C_VEL
LIN {X 0,Y 256.563,Z 788.844,A -85,B 0,C 180,E1 12771.483,E2 12771.483} C_VEL
LIN {X 0,Y 257.259,Z 781.522,A -85,B 0,C 180,E1 12767.657,E2 12767.657} C_VEL
LIN {X 0,Y 258.431,Z 772.749,A -85,B 0,C 180,E1 12764.056,E2 12764.056} C_VEL
LIN {X 0,Y 260.069,Z 762.612,A -85,B 0,C 180,E1 12760.692,E2 12760.692} C_VEL
LIN {X 0,Y 262.363,Z 749.902,A -85,B 0,C 180,E1 12757.259,E2 12757.259} C_VEL
LIN {X 0,Y 265.026,Z 735.894,A -85,B 0,C 180,E1 12754.167,E2 12754.167} C_VEL
LIN {X 0,Y 267.95,Z 720.552,A -85,B 0,C 180,E1 12751.388,E2 12751.388} C_VEL
LIN {X 0,Y 271.015,Z 703.628,A -85,B 0,C 180,E1 12748.902,E2 12748.902} C_VEL
LIN {X 0,Y 274.121,Z 685.075,A -85,B 0,C 180,E1 12746.705,E2 12746.705} C_VEL
LIN {X 0,Y 276.884,Z 666.498,A -85,B 0,C 180,E1 12744.958,E2 12744.958} C_VEL
LIN {X 0,Y 279.316,Z 647.054,A -85,B 0,C 180,E1 12743.542,E2 12743.542} C_VEL
LIN {X 0,Y 281.323,Z 626.353,A -85,B 0,C 180,E1 12742.45,E2 12742.45} C_VEL
LIN {X 0,Y 293.595,Z 469.131,A -85,B 0,C 180,E1 12736.884,E2 12736.884} C_VEL
LIN {X 0,Y 280.86,Z 442.271,A -85,B 0,C 180,E1 12734.034,E2 12734.034} C_VEL
LIN {X 0,Y 268.375,Z 418.078,A -85,B 0,C 180,E1 12731.044,E2 12731.044} C_VEL
LIN {X 0,Y 265.74,Z 411.804,A -85,B 0,C 180,E1 12729.765,E2 12729.765} C_VEL
LIN {X 0,Y 259.79,Z 397.962,A -85,B 0,C 180,E1 12726.624,E2 12726.624} C_VEL
LIN {X 0,Y 258.551,Z 394.592,A -85,B 0,C 180,E1 12725.831,E2 12725.831} C_VEL
LIN {X 0,Y 258.558,Z 394.594,A -85,B 0,C 180,E1 12720.694,E2 12720.694} C_VEL
LIN {X 0,Y 258.557,Z 394.591,A -85,B 0,C 180,E1 12715.911,E2 12715.911} C_VEL
LIN {X 0,Y 258.546,Z 394.587,A -85,B 0,C 180,E1 12710.842,E2 12710.842} C_VEL
LIN {X 0,Y 258.563,Z 394.591,A -85,B 0,C 180,E1 12705.936,E2 12705.936} C_VEL
LIN {X 0,Y 258.541,Z 394.594,A -85,B 0,C 180,E1 12701.149,E2 12701.149} C_VEL
LIN {X 0,Y 258.565,Z 394.591,A -85,B 0,C 180,E1 12696.216,E2 12696.216} C_VEL
LIN {X 0,Y 258.543,Z 394.592,A -85,B 0,C 180,E1 12691.33,E2 12691.33} C_VEL
LIN {X 0,Y 258.546,Z 394.586,A -85,B 0,C 180,E1 12686.452,E2 12686.452} C_VEL
LIN {X 0,Y 258.566,Z 394.582,A -85,B 0,C 180,E1 12681.774,E2 12681.774} C_VEL
LIN {X 0,Y 258.538,Z 394.59,A -85,B 0,C 180,E1 12676.81,E2 12676.81} C_VEL
LIN {X 0,Y 258.559,Z 394.591,A -85,B 0,C 180,E1 12671.979,E2 12671.979} C_VEL
LIN {X 0,Y 258.552,Z 394.592,A -85,B 0,C 180,E1 12667.25,E2 12667.25} C_VEL
LIN {X 0,Y 258.554,Z 394.591,A -85,B 0,C 180,E1 12662.1,E2 12662.1} C_VEL
LIN {X 0,Y 258.559,Z 394.594,A -85,B 0,C 180,E1 12657.46,E2 12657.46} C_VEL
LIN {X 0,Y 258.538,Z 394.6,A -85,B 0,C 180,E1 12652.449,E2 12652.449} C_VEL
LIN {X 0,Y 258.573,Z 394.818,A -85,B 0,C 180,E1 12650.211,E2 12650.211} C_VEL
LIN {X 0,Y 263.127,Z 409.596,A -85,B 0,C 180,E1 12645.638,E2 12645.638} C_VEL
LIN {X 0,Y 267.457,Z 424.857,A -85,B 0,C 180,E1 12641.286,E2 12641.286} C_VEL
LIN {X 0,Y 271.688,Z 441.664,A -85,B 0,C 180,E1 12636.861,E2 12636.861} C_VEL
LIN {X 0,Y 273.19,Z 448.901,A -85,B 0,C 180,E1 12635.073,E2 12635.073} C_VEL
LIN {X 0,Y 268.694,Z 474.256,A -85,B 0,C 180,E1 12629.883,E2 12629.883} C_VEL
LIN {X 0,Y 268.344,Z 476.947,A -85,B 0,C 180,E1 12629.413,E2 12629.413} C_VEL
LIN {X 0,Y 271.924,Z 519.294,A -85,B 0,C 180,E1 12627.185,E2 12627.185} C_VEL
LIN {X 0,Y 268.259,Z 577.208,A -85,B 0,C 180,E1 12624.776,E2 12624.776} C_VEL
LIN {X 0,Y 266.885,Z 584.752,A -85,B 0,C 180,E1 12624.514,E2 12624.514} C_VEL
LIN {X 0,Y 259.749,Z 604.602,A -85,B 0,C 180,E1 12623.969,E2 12623.969} C_VEL
LIN {X 0,Y 258.711,Z 611.052,A -85,B 0,C 180,E1 12623.694,E2 12623.694} C_VEL
LIN {X 0,Y 257.594,Z 630.184,A -85,B 0,C 180,E1 12622.479,E2 12622.479} C_VEL
LIN {X 0,Y 256.167,Z 648.922,A -85,B 0,C 180,E1 12620.805,E2 12620.805} C_VEL
LIN {X 0,Y 254.652,Z 666.02,A -85,B 0,C 180,E1 12618.782,E2 12618.782} C_VEL
LIN {X 0,Y 253.231,Z 681.924,A -85,B 0,C 180,E1 12616.369,E2 12616.369} C_VEL
LIN {X 0,Y 251.971,Z 696.06,A -85,B 0,C 180,E1 12613.657,E2 12613.657} C_VEL
LIN {X 0,Y 250.991,Z 708.794,A -85,B 0,C 180,E1 12610.559,E2 12610.559} C_VEL
LIN {X 0,Y 250.432,Z 719.211,A -85,B 0,C 180,E1 12607.341,E2 12607.341} C_VEL
LIN {X 0,Y 250.306,Z 726.855,A -85,B 0,C 180,E1 12604.353,E2 12604.353} C_VEL
LIN {X 0,Y 250.603,Z 733.507,A -85,B 0,C 180,E1 12600.915,E2 12600.915} C_VEL
LIN {X 0,Y 251.325,Z 737.916,A -85,B 0,C 180,E1 12597.72,E2 12597.72} C_VEL
LIN {X 0,Y 252.786,Z 740.985,A -85,B 0,C 180,E1 12594.098,E2 12594.098} C_VEL
LIN {X 0,Y 254.83,Z 742.006,A -85,B 0,C 180,E1 12590.743,E2 12590.743} C_VEL
LIN {X 0,Y 257.81,Z 741.192,A -85,B 0,C 180,E1 12587.229,E2 12587.229} C_VEL
LIN {X 0,Y 261.359,Z 738.672,A -85,B 0,C 180,E1 12584.012,E2 12584.012} C_VEL
LIN {X 0,Y 265.959,Z 734.017,A -85,B 0,C 180,E1 12580.681,E2 12580.681} C_VEL
LIN {X 0,Y 271.069,Z 727.826,A -85,B 0,C 180,E1 12577.671,E2 12577.671} C_VEL
LIN {X 0,Y 277.361,Z 719.095,A -85,B 0,C 180,E1 12574.597,E2 12574.597} C_VEL
LIN {X 0,Y 284.49,Z 707.89,A -85,B 0,C 180,E1 12571.676,E2 12571.676} C_VEL
LIN {X 0,Y 291.46,Z 695.707,A -85,B 0,C 180,E1 12569.26,E2 12569.26} C_VEL
LIN {X 0,Y 298.295,Z 682.54,A -85,B 0,C 180,E1 12567.226,E2 12567.226} C_VEL
LIN {X 0,Y 305.358,Z 667.181,A -85,B 0,C 180,E1 12565.382,E2 12565.382} C_VEL
LIN {X 0,Y 311.29,Z 652.248,A -85,B 0,C 180,E1 12564,E2 12564} C_VEL
LIN {X 0,Y 316.861,Z 635.534,A -85,B 0,C 180,E1 12562.823,E2 12562.823} C_VEL
LIN {X 0,Y 325.425,Z 604.078,A -85,B 0,C 180,E1 12561.243,E2 12561.243} C_VEL
LIN {X 0,Y 335.105,Z 569.186,A -85,B 0,C 180,E1 12559.705,E2 12559.705} C_VEL
LIN {X 0,Y 319.454,Z 630.632,A -85,B 0,C 180,E1 12557.402,E2 12557.402} C_VEL
LIN {X 0,Y 313.244,Z 653.47,A -85,B 0,C 180,E1 12556.434,E2 12556.434} C_VEL
LIN {X 0,Y 306.489,Z 672.992,A -85,B 0,C 180,E1 12555.332,E2 12555.332} C_VEL
LIN {X 0,Y 299.096,Z 691.386,A -85,B 0,C 180,E1 12553.921,E2 12553.921} C_VEL
LIN {X 0,Y 291.907,Z 707.33,A -85,B 0,C 180,E1 12552.304,E2 12552.304} C_VEL
LIN {X 0,Y 284.396,Z 722.826,A -85,B 0,C 180,E1 12550.279,E2 12550.279} C_VEL
LIN {X 0,Y 276.986,Z 737.411,A -85,B 0,C 180,E1 12547.855,E2 12547.855} C_VEL
LIN {X 0,Y 269.98,Z 750.91,A -85,B 0,C 180,E1 12545.032,E2 12545.032} C_VEL
LIN {X 0,Y 263.626,Z 763.215,A -85,B 0,C 180,E1 12541.816,E2 12541.816} C_VEL
LIN {X 0,Y 258.161,Z 774.258,A -85,B 0,C 180,E1 12538.197,E2 12538.197} C_VEL
LIN {X 0,Y 253.844,Z 783.961,A -85,B 0,C 180,E1 12534.183,E2 12534.183} C_VEL
LIN {X 0,Y 250.921,Z 792.243,A -85,B 0,C 180,E1 12529.798,E2 12529.798} C_VEL
LIN {X 0,Y 250.605,Z 793.687,A -85,B 0,C 180,E1 12529.097,E2 12529.097} C_VEL
LIN {X 0,Y 249.301,Z 804.014,A -85,B 0,C 180,E1 12525.349,E2 12525.349} C_VEL
LIN {X 0,Y 248.643,Z 812.18,A -85,B 0,C 180,E1 12521.599,E2 12521.599} C_VEL
LIN {X 0,Y 248.521,Z 818.447,A -85,B 0,C 180,E1 12517.862,E2 12517.862} C_VEL
LIN {X 0,Y 248.642,Z 822.942,A -85,B 0,C 180,E1 12514.151,E2 12514.151} C_VEL
LIN {X 0,Y 248.698,Z 825.601,A -85,B 0,C 180,E1 12510.691,E2 12510.691} C_VEL
LIN {X 0,Y 248.474,Z 826.92,A -85,B 0,C 180,E1 12507.001,E2 12507.001} C_VEL
LIN {X 0,Y 248.222,Z 826.748,A -85,B 0,C 180,E1 12503.059,E2 12503.059} C_VEL
LIN {X 0,Y 248.384,Z 824.894,A -85,B 0,C 180,E1 12498.859,E2 12498.859} C_VEL
LIN {X 0,Y 249.546,Z 821.166,A -85,B 0,C 180,E1 12494.428,E2 12494.428} C_VEL
LIN {X 0,Y 251.952,Z 815.649,A -85,B 0,C 180,E1 12490.045,E2 12490.045} C_VEL
LIN {X 0,Y 256.034,Z 807.888,A -85,B 0,C 180,E1 12485.547,E2 12485.547} C_VEL
LIN {X 0,Y 261.763,Z 798.085,A -85,B 0,C 180,E1 12481.231,E2 12481.231} C_VEL
LIN {X 0,Y 268.787,Z 786.809,A -85,B 0,C 180,E1 12477.358,E2 12477.358} C_VEL
LIN {X 0,Y 277.362,Z 773.513,A -85,B 0,C 180,E1 12473.757,E2 12473.757} C_VEL
LIN {X 0,Y 286.912,Z 758.851,A -85,B 0,C 180,E1 12470.635,E2 12470.635} C_VEL
LIN {X 0,Y 297.552,Z 742.461,A -85,B 0,C 180,E1 12467.904,E2 12467.904} C_VEL
LIN {X 0,Y 308.482,Z 725.279,A -85,B 0,C 180,E1 12465.694,E2 12465.694} C_VEL
LIN {X 0,Y 318.437,Z 708.941,A -85,B 0,C 180,E1 12464.056,E2 12464.056} C_VEL
LIN {X 0,Y 307.911,Z 725.258,A -85,B 0,C 180,E1 12461.984,E2 12461.984} C_VEL
LIN {X 0,Y 297.367,Z 740.631,A -85,B 0,C 180,E1 12459.456,E2 12459.456} C_VEL
LIN {X 0,Y 287.369,Z 754.545,A -85,B 0,C 180,E1 12456.51,E2 12456.51} C_VEL
LIN {X 0,Y 278.12,Z 767.047,A -85,B 0,C 180,E1 12453.124,E2 12453.124} C_VEL
LIN {X 0,Y 270.17,Z 777.398,A -85,B 0,C 180,E1 12449.486,E2 12449.486} C_VEL
LIN {X 0,Y 263.53,Z 785.788,A -85,B 0,C 180,E1 12445.628,E2 12445.628} C_VEL
LIN {X 0,Y 257.955,Z 792.64,A -85,B 0,C 180,E1 12441.367,E2 12441.367} C_VEL
LIN {X 0,Y 253.971,Z 797.342,A -85,B 0,C 180,E1 12437.173,E2 12437.173} C_VEL
LIN {X 0,Y 251.194,Z 800.311,A -85,B 0,C 180,E1 12432.879,E2 12432.879} C_VEL
LIN {X 0,Y 249.477,Z 801.563,A -85,B 0,C 180,E1 12428.528,E2 12428.528} C_VEL
LIN {X 0,Y 248.638,Z 801.121,A -85,B 0,C 180,E1 12424.382,E2 12424.382} C_VEL
LIN {X 0,Y 248.314,Z 799.206,A -85,B 0,C 180,E1 12420.461,E2 12420.461} C_VEL
LIN {X 0,Y 248.248,Z 795.773,A -85,B 0,C 180,E1 12416.536,E2 12416.536} C_VEL
LIN {X 0,Y 248.444,Z 790.695,A -85,B 0,C 180,E1 12412.6,E2 12412.6} C_VEL
LIN {X 0,Y 249.027,Z 783.812,A -85,B 0,C 180,E1 12408.653,E2 12408.653} C_VEL
LIN {X 0,Y 250.067,Z 775.497,A -85,B 0,C 180,E1 12404.936,E2 12404.936} C_VEL
LIN {X 0,Y 251.711,Z 765.149,A -85,B 0,C 180,E1 12401.231,E2 12401.231} C_VEL
LIN {X 0,Y 253.899,Z 753.068,A -85,B 0,C 180,E1 12397.735,E2 12397.735} C_VEL
LIN {X 0,Y 256.554,Z 739.319,A -85,B 0,C 180,E1 12394.491,E2 12394.491} C_VEL
LIN {X 0,Y 259.611,Z 723.671,A -85,B 0,C 180,E1 12391.473,E2 12391.473} C_VEL
LIN {X 0,Y 262.785,Z 706.904,A -85,B 0,C 180,E1 12388.838,E2 12388.838} C_VEL
LIN {X 0,Y 265.904,Z 689.156,A -85,B 0,C 180,E1 12386.592,E2 12386.592} C_VEL
LIN {X 0,Y 268.893,Z 670.047,A -85,B 0,C 180,E1 12384.674,E2 12384.674} C_VEL
LIN {X 0,Y 271.537,Z 650.028,A -85,B 0,C 180,E1 12383.115,E2 12383.115} C_VEL
LIN {X 0,Y 273.714,Z 629.519,A -85,B 0,C 180,E1 12381.935,E2 12381.935} C_VEL
LIN {X 0,Y 280.773,Z 540.391,A -85,B 0,C 180,E1 12378.587,E2 12378.587} C_VEL
LIN {X 0,Y 286.568,Z 471.425,A -85,B 0,C 180,E1 12376.132,E2 12376.132} C_VEL
LIN {X 0,Y 272.911,Z 442.688,A -85,B 0,C 180,E1 12372.957,E2 12372.957} C_VEL
LIN {X 0,Y 259.885,Z 417.671,A -85,B 0,C 180,E1 12369.692,E2 12369.692} C_VEL
LIN {X 0,Y 253.566,Z 402.735,A -85,B 0,C 180,E1 12366.262,E2 12366.262} C_VEL
LIN {X 0,Y 250.677,Z 395.98,A -85,B 0,C 180,E1 12364.638,E2 12364.638} C_VEL
LIN {X 0,Y 250.622,Z 395.58,A -85,B 0,C 180,E1 12364.507,E2 12364.507} C_VEL
LIN {X 0,Y 250.606,Z 395.579,A -85,B 0,C 180,E1 12359.567,E2 12359.567} C_VEL
LIN {X 0,Y 250.621,Z 395.577,A -85,B 0,C 180,E1 12354.514,E2 12354.514} C_VEL
LIN {X 0,Y 250.615,Z 395.58,A -85,B 0,C 180,E1 12349.685,E2 12349.685} C_VEL
LIN {X 0,Y 250.612,Z 395.583,A -85,B 0,C 180,E1 12344.557,E2 12344.557} C_VEL
LIN {X 0,Y 250.612,Z 395.576,A -85,B 0,C 180,E1 12339.646,E2 12339.646} C_VEL
LIN {X 0,Y 250.606,Z 395.575,A -85,B 0,C 180,E1 12334.577,E2 12334.577} C_VEL
LIN {X 0,Y 250.625,Z 395.574,A -85,B 0,C 180,E1 12329.771,E2 12329.771} C_VEL
LIN {X 0,Y 250.6,Z 395.581,A -85,B 0,C 180,E1 12324.735,E2 12324.735} C_VEL
LIN {X 0,Y 250.622,Z 395.581,A -85,B 0,C 180,E1 12319.89,E2 12319.89} C_VEL
LIN {X 0,Y 250.601,Z 395.584,A -85,B 0,C 180,E1 12314.917,E2 12314.917} C_VEL
LIN {X 0,Y 250.622,Z 395.579,A -85,B 0,C 180,E1 12309.934,E2 12309.934} C_VEL
LIN {X 0,Y 250.612,Z 395.579,A -85,B 0,C 180,E1 12305.234,E2 12305.234} C_VEL
LIN {X 0,Y 250.613,Z 395.579,A -85,B 0,C 180,E1 12300.085,E2 12300.085} C_VEL
LIN {X 0,Y 250.61,Z 395.586,A -85,B 0,C 180,E1 12295.213,E2 12295.213} C_VEL
LIN {X 0,Y 250.656,Z 395.827,A -85,B 0,C 180,E1 12291.298,E2 12291.298} C_VEL
LIN {X 0,Y 255.234,Z 410.545,A -85,B 0,C 180,E1 12286.567,E2 12286.567} C_VEL
LIN {X 0,Y 259.612,Z 426.106,A -85,B 0,C 180,E1 12281.985,E2 12281.985} C_VEL
LIN {X 0,Y 263.452,Z 441.202,A -85,B 0,C 180,E1 12277.869,E2 12277.869} C_VEL
LIN {X 0,Y 265.503,Z 450.674,A -85,B 0,C 180,E1 12275.447,E2 12275.447} C_VEL
LIN {X 0,Y 260.798,Z 476.356,A -85,B 0,C 180,E1 12270.077,E2 12270.077} C_VEL
LIN {X 0,Y 264.294,Z 520.076,A -85,B 0,C 180,E1 12267.701,E2 12267.701} C_VEL
LIN {X 0,Y 258.711,Z 611.052,A -85,B 0,C 180,E1 12263.694,E2 12263.694} C_VEL
LIN {X 0,Y 257.365,Z 618.533,A -85,B 0,C 180,E1 12263.336,E2 12263.336} C_VEL
LIN {X 0,Y 250.991,Z 634.796,A -85,B 0,C 180,E1 12262.435,E2 12262.435} C_VEL
LIN {X 0,Y 248.996,Z 641.892,A -85,B 0,C 180,E1 12261.858,E2 12261.858} C_VEL
LIN {X 0,Y 248.736,Z 643.929,A -85,B 0,C 180,E1 12261.661,E2 12261.661} C_VEL
LIN {X 0,Y 247.217,Z 661.176,A -85,B 0,C 180,E1 12259.738,E2 12259.738} C_VEL
LIN {X 0,Y 245.74,Z 677.329,A -85,B 0,C 180,E1 12257.401,E2 12257.401} C_VEL
LIN {X 0,Y 244.368,Z 692.136,A -85,B 0,C 180,E1 12254.696,E2 12254.696} C_VEL
LIN {X 0,Y 243.33,Z 704.57,A -85,B 0,C 180,E1 12251.856,E2 12251.856} C_VEL
LIN {X 0,Y 242.667,Z 714.736,A -85,B 0,C 180,E1 12249.008,E2 12249.008} C_VEL
LIN {X 0,Y 242.326,Z 724.162,A -85,B 0,C 180,E1 12245.683,E2 12245.683} C_VEL
LIN {X 0,Y 242.43,Z 731.43,A -85,B 0,C 180,E1 12242.364,E2 12242.364} C_VEL
LIN {X 0,Y 243.053,Z 737.261,A -85,B 0,C 180,E1 12238.822,E2 12238.822} C_VEL
LIN {X 0,Y 244.349,Z 741.289,A -85,B 0,C 180,E1 12235.071,E2 12235.071} C_VEL
LIN {X 0,Y 246.286,Z 743.292,A -85,B 0,C 180,E1 12231.596,E2 12231.596} C_VEL
LIN {X 0,Y 248.953,Z 743.491,A -85,B 0,C 180,E1 12228.181,E2 12228.181} C_VEL
LIN {X 0,Y 252.661,Z 741.909,A -85,B 0,C 180,E1 12224.625,E2 12224.625} C_VEL
LIN {X 0,Y 257.252,Z 738.357,A -85,B 0,C 180,E1 12221.18,E2 12221.18} C_VEL
LIN {X 0,Y 262.758,Z 732.911,A -85,B 0,C 180,E1 12217.87,E2 12217.87} C_VEL
LIN {X 0,Y 269.57,Z 724.816,A -85,B 0,C 180,E1 12214.517,E2 12214.517} C_VEL
LIN {X 0,Y 276.405,Z 715.588,A -85,B 0,C 180,E1 12211.714,E2 12211.714} C_VEL
LIN {X 0,Y 284.04,Z 704.221,A -85,B 0,C 180,E1 12209.074,E2 12209.074} C_VEL
LIN {X 0,Y 292.186,Z 690.646,A -85,B 0,C 180,E1 12206.686,E2 12206.686} C_VEL
LIN {X 0,Y 300.097,Z 675.697,A -85,B 0,C 180,E1 12204.686,E2 12204.686} C_VEL
LIN {X 0,Y 306.921,Z 661.02,A -85,B 0,C 180,E1 12203.172,E2 12203.172} C_VEL
LIN {X 0,Y 313.381,Z 644.498,A -85,B 0,C 180,E1 12201.876,E2 12201.876} C_VEL
LIN {X 0,Y 319.02,Z 626.53,A -85,B 0,C 180,E1 12200.837,E2 12200.837} C_VEL
LIN {X 0,Y 325.169,Z 604.839,A -85,B 0,C 180,E1 12199.811,E2 12199.811} C_VEL
LIN {X 0,Y 314.219,Z 645.253,A -85,B 0,C 180,E1 12198.262,E2 12198.262} C_VEL
LIN {X 0,Y 307.071,Z 665.768,A -85,B 0,C 180,E1 12197.245,E2 12197.245} C_VEL
LIN {X 0,Y 299.489,Z 684.048,A -85,B 0,C 180,E1 12196.01,E2 12196.01} C_VEL
LIN {X 0,Y 290.99,Z 702.019,A -85,B 0,C 180,E1 12194.366,E2 12194.366} C_VEL
LIN {X 0,Y 282.592,Z 718.308,A -85,B 0,C 180,E1 12192.379,E2 12192.379} C_VEL
LIN {X 0,Y 274.108,Z 733.627,A -85,B 0,C 180,E1 12189.941,E2 12189.941} C_VEL
LIN {X 0,Y 265.861,Z 748.031,A -85,B 0,C 180,E1 12186.995,E2 12186.995} C_VEL
LIN {X 0,Y 258.801,Z 760.322,A -85,B 0,C 180,E1 12183.803,E2 12183.803} C_VEL
LIN {X 0,Y 252.603,Z 771.441,A -85,B 0,C 180,E1 12180.179,E2 12180.179} C_VEL
LIN {X 0,Y 247.528,Z 781.27,A -85,B 0,C 180,E1 12176.123,E2 12176.123} C_VEL
LIN {X 0,Y 243.866,Z 789.68,A -85,B 0,C 180,E1 12171.654,E2 12171.654} C_VEL
LIN {X 0,Y 242.549,Z 793.74,A -85,B 0,C 180,E1 12169.006,E2 12169.006} C_VEL
LIN {X 0,Y 241.269,Z 803.934,A -85,B 0,C 180,E1 12165.134,E2 12165.134} C_VEL
LIN {X 0,Y 240.651,Z 811.996,A -85,B 0,C 180,E1 12161.261,E2 12161.261} C_VEL
LIN {X 0,Y 240.58,Z 818.161,A -85,B 0,C 180,E1 12157.402,E2 12157.402} C_VEL
LIN {X 0,Y 240.7,Z 822.34,A -85,B 0,C 180,E1 12153.811,E2 12153.811} C_VEL
LIN {X 0,Y 240.734,Z 824.984,A -85,B 0,C 180,E1 12150.238,E2 12150.238} C_VEL
LIN {X 0,Y 240.456,Z 826.302,A -85,B 0,C 180,E1 12146.424,E2 12146.424} C_VEL
LIN {X 0,Y 240.205,Z 826.102,A -85,B 0,C 180,E1 12142.171,E2 12142.171} C_VEL
LIN {X 0,Y 240.603,Z 824.035,A -85,B 0,C 180,E1 12137.52,E2 12137.52} C_VEL
LIN {X 0,Y 242.28,Z 819.965,A -85,B 0,C 180,E1 12132.714,E2 12132.714} C_VEL
LIN {X 0,Y 245.492,Z 813.977,A -85,B 0,C 180,E1 12127.994,E2 12127.994} C_VEL
LIN {X 0,Y 250.392,Z 806.068,A -85,B 0,C 180,E1 12123.433,E2 12123.433} C_VEL
LIN {X 0,Y 257.023,Z 796.206,A -85,B 0,C 180,E1 12119.103,E2 12119.103} C_VEL
LIN {X 0,Y 265.41,Z 784.333,A -85,B 0,C 180,E1 12115.067,E2 12115.067} C_VEL
LIN {X 0,Y 274.98,Z 771.037,A -85,B 0,C 180,E1 12111.554,E2 12111.554} C_VEL
LIN {X 0,Y 286.104,Z 755.693,A -85,B 0,C 180,E1 12108.394,E2 12108.394} C_VEL
LIN {X 0,Y 297.395,Z 739.995,A -85,B 0,C 180,E1 12105.897,E2 12105.897} C_VEL
LIN {X 0,Y 308.588,Z 723.979,A -85,B 0,C 180,E1 12103.898,E2 12103.898} C_VEL
LIN {X 0,Y 297.147,Z 739.263,A -85,B 0,C 180,E1 12101.52,E2 12101.52} C_VEL
LIN {X 0,Y 286.195,Z 753.186,A -85,B 0,C 180,E1 12098.708,E2 12098.708} C_VEL
LIN {X 0,Y 275.917,Z 765.675,A -85,B 0,C 180,E1 12095.436,E2 12095.436} C_VEL
LIN {X 0,Y 266.552,Z 776.706,A -85,B 0,C 180,E1 12091.678,E2 12091.678} C_VEL
LIN {X 0,Y 258.681,Z 785.678,A -85,B 0,C 180,E1 12087.634,E2 12087.634} C_VEL
LIN {X 0,Y 252.297,Z 792.618,A -85,B 0,C 180,E1 12083.347,E2 12083.347} C_VEL
LIN {X 0,Y 247.407,Z 797.67,A -85,B 0,C 180,E1 12078.863,E2 12078.863} C_VEL
LIN {X 0,Y 243.953,Z 800.859,A -85,B 0,C 180,E1 12074.236,E2 12074.236} C_VEL
LIN {X 0,Y 241.876,Z 802.168,A -85,B 0,C 180,E1 12069.758,E2 12069.758} C_VEL
LIN {X 0,Y 240.802,Z 801.815,A -85,B 0,C 180,E1 12065.48,E2 12065.48} C_VEL
LIN {X 0,Y 240.355,Z 799.863,A -85,B 0,C 180,E1 12061.192,E2 12061.192} C_VEL
LIN {X 0,Y 240.245,Z 796.47,A -85,B 0,C 180,E1 12057.137,E2 12057.137} C_VEL
LIN {X 0,Y 240.398,Z 791.445,A -85,B 0,C 180,E1 12053.072,E2 12053.072} C_VEL
LIN {X 0,Y 240.95,Z 784.625,A -85,B 0,C 180,E1 12048.995,E2 12048.995} C_VEL
LIN {X 0,Y 241.967,Z 776.377,A -85,B 0,C 180,E1 12045.155,E2 12045.155} C_VEL
LIN {X 0,Y 243.601,Z 766.099,A -85,B 0,C 180,E1 12041.328,E2 12041.328} C_VEL
LIN {X 0,Y 245.767,Z 754.328,A -85,B 0,C 180,E1 12037.768,E2 12037.768} C_VEL
LIN {X 0,Y 248.392,Z 741.049,A -85,B 0,C 180,E1 12034.487,E2 12034.487} C_VEL
LIN {X 0,Y 251.358,Z 726.259,A -85,B 0,C 180,E1 12031.488,E2 12031.488} C_VEL
LIN {X 0,Y 254.7,Z 709.118,A -85,B 0,C 180,E1 12028.657,E2 12028.657} C_VEL
LIN {X 0,Y 257.889,Z 691.686,A -85,B 0,C 180,E1 12026.329,E2 12026.329} C_VEL
LIN {X 0,Y 260.905,Z 673.397,A -85,B 0,C 180,E1 12024.373,E2 12024.373} C_VEL
LIN {X 0,Y 263.683,Z 653.551,A -85,B 0,C 180,E1 12022.723,E2 12022.723} C_VEL
LIN {X 0,Y 266.069,Z 632.553,A -85,B 0,C 180,E1 12021.422,E2 12021.422} C_VEL
LIN {X 0,Y 268.357,Z 605.131,A -85,B 0,C 180,E1 12020.257,E2 12020.257} C_VEL
LIN {X 0,Y 279.603,Z 473.854,A -85,B 0,C 180,E1 12015.367,E2 12015.367} C_VEL
LIN {X 0,Y 266.503,Z 446.29,A -85,B 0,C 180,E1 12012.225,E2 12012.225} C_VEL
LIN {X 0,Y 253.72,Z 421.566,A -85,B 0,C 180,E1 12008.908,E2 12008.908} C_VEL
LIN {X 0,Y 251.664,Z 417.674,A -85,B 0,C 180,E1 12008.301,E2 12008.301} C_VEL
LIN {X 0,Y 244.218,Z 400.376,A -85,B 0,C 180,E1 12004.118,E2 12004.118} C_VEL
LIN {X 0,Y 242.701,Z 396.823,A -85,B 0,C 180,E1 12003.225,E2 12003.225} C_VEL
LIN {X 0,Y 242.694,Z 396.569,A -85,B 0,C 180,E1 11998.28,E2 11998.28} C_VEL
LIN {X 0,Y 242.665,Z 396.568,A -85,B 0,C 180,E1 11993.044,E2 11993.044} C_VEL
LIN {X 0,Y 242.683,Z 396.565,A -85,B 0,C 180,E1 11987.999,E2 11987.999} C_VEL
LIN {X 0,Y 242.664,Z 396.563,A -85,B 0,C 180,E1 11982.856,E2 11982.856} C_VEL
LIN {X 0,Y 242.684,Z 396.562,A -85,B 0,C 180,E1 11977.814,E2 11977.814} C_VEL
LIN {X 0,Y 242.665,Z 396.563,A -85,B 0,C 180,E1 11972.598,E2 11972.598} C_VEL
LIN {X 0,Y 242.68,Z 396.556,A -85,B 0,C 180,E1 11967.875,E2 11967.875} C_VEL
LIN {X 0,Y 242.661,Z 396.562,A -85,B 0,C 180,E1 11962.661,E2 11962.661} C_VEL
LIN {X 0,Y 242.679,Z 396.563,A -85,B 0,C 180,E1 11957.629,E2 11957.629} C_VEL
LIN {X 0,Y 242.665,Z 396.568,A -85,B 0,C 180,E1 11952.495,E2 11952.495} C_VEL
LIN {X 0,Y 242.684,Z 396.57,A -85,B 0,C 180,E1 11947.47,E2 11947.47} C_VEL
LIN {X 0,Y 242.67,Z 396.569,A -85,B 0,C 180,E1 11942.252,E2 11942.252} C_VEL
LIN {X 0,Y 242.678,Z 396.573,A -85,B 0,C 180,E1 11937.334,E2 11937.334} C_VEL
LIN {X 0,Y 242.668,Z 396.631,A -85,B 0,C 180,E1 11932.507,E2 11932.507} C_VEL
LIN {X 0,Y 246.92,Z 410.334,A -85,B 0,C 180,E1 11927.92,E2 11927.92} C_VEL
LIN {X 0,Y 251.168,Z 424.97,A -85,B 0,C 180,E1 11923.406,E2 11923.406} C_VEL
LIN {X 0,Y 255.341,Z 441.235,A -85,B 0,C 180,E1 11918.795,E2 11918.795} C_VEL
LIN {X 0,Y 257.821,Z 452.36,A -85,B 0,C 180,E1 11915.845,E2 11915.845} C_VEL
LIN {X 0,Y 253.284,Z 476.628,A -85,B 0,C 180,E1 11910.709,E2 11910.709} C_VEL
LIN {X 0,Y 256.656,Z 520.822,A -85,B 0,C 180,E1 11908.227,E2 11908.227} C_VEL
LIN {X 0,Y 250.725,Z 614.577,A -85,B 0,C 180,E1 11903.904,E2 11903.904} C_VEL
LIN {X 0,Y 249.564,Z 633.154,A -85,B 0,C 180,E1 11902.62,E2 11902.62} C_VEL
LIN {X 0,Y 248.736,Z 643.929,A -85,B 0,C 180,E1 11901.661,E2 11901.661} C_VEL
LIN {X 0,Y 247.166,Z 650.997,A -85,B 0,C 180,E1 11900.975,E2 11900.975} C_VEL
LIN {X 0,Y 239.703,Z 667.86,A -85,B 0,C 180,E1 11899.098,E2 11899.098} C_VEL
LIN {X 0,Y 238.095,Z 674.333,A -85,B 0,C 180,E1 11898.142,E2 11898.142} C_VEL
LIN {X 0,Y 236.72,Z 688.926,A -85,B 0,C 180,E1 11895.571,E2 11895.571} C_VEL
LIN {X 0,Y 235.508,Z 702.819,A -85,B 0,C 180,E1 11892.505,E2 11892.505} C_VEL
LIN {X 0,Y 234.673,Z 715.039,A -85,B 0,C 180,E1 11889.071,E2 11889.071} C_VEL
LIN {X 0,Y 234.329,Z 724.666,A -85,B 0,C 180,E1 11885.632,E2 11885.632} C_VEL
LIN {X 0,Y 234.459,Z 732.206,A -85,B 0,C 180,E1 11882.2,E2 11882.2} C_VEL
LIN {X 0,Y 235.201,Z 738.537,A -85,B 0,C 180,E1 11878.295,E2 11878.295} C_VEL
LIN {X 0,Y 236.555,Z 742.49,A -85,B 0,C 180,E1 11874.665,E2 11874.665} C_VEL
LIN {X 0,Y 238.814,Z 744.814,A -85,B 0,C 180,E1 11870.846,E2 11870.846} C_VEL
LIN {X 0,Y 241.977,Z 745.139,A -85,B 0,C 180,E1 11867.107,E2 11867.107} C_VEL
LIN {X 0,Y 246.074,Z 743.625,A -85,B 0,C 180,E1 11863.476,E2 11863.476} C_VEL
LIN {X 0,Y 251.105,Z 740.211,A -85,B 0,C 180,E1 11859.975,E2 11859.975} C_VEL
LIN {X 0,Y 257.487,Z 734.562,A -85,B 0,C 180,E1 11856.424,E2 11856.424} C_VEL
LIN {X 0,Y 264.894,Z 726.621,A -85,B 0,C 180,E1 11853.067,E2 11853.067} C_VEL
LIN {X 0,Y 272.268,Z 717.614,A -85,B 0,C 180,E1 11850.28,E2 11850.28} C_VEL
LIN {X 0,Y 280.465,Z 706.578,A -85,B 0,C 180,E1 11847.673,E2 11847.673} C_VEL
LIN {X 0,Y 289.455,Z 692.928,A -85,B 0,C 180,E1 11845.253,E2 11845.253} C_VEL
LIN {X 0,Y 297.532,Z 679.059,A -85,B 0,C 180,E1 11843.381,E2 11843.381} C_VEL
LIN {X 0,Y 305.069,Z 664.275,A -85,B 0,C 180,E1 11841.844,E2 11841.844} C_VEL
LIN {X 0,Y 311.784,Z 648.737,A -85,B 0,C 180,E1 11840.612,E2 11840.612} C_VEL
LIN {X 0,Y 315.346,Z 639.04,A -85,B 0,C 180,E1 11839.989,E2 11839.989} C_VEL
LIN {X 0,Y 308.232,Z 659.22,A -85,B 0,C 180,E1 11839.097,E2 11839.097} C_VEL
LIN {X 0,Y 300.153,Z 678.034,A -85,B 0,C 180,E1 11837.975,E2 11837.975} C_VEL
LIN {X 0,Y 291.795,Z 695.097,A -85,B 0,C 180,E1 11836.589,E2 11836.589} C_VEL
LIN {X 0,Y 283.28,Z 710.698,A -85,B 0,C 180,E1 11834.904,E2 11834.904} C_VEL
LIN {X 0,Y 274.182,Z 726.18,A -85,B 0,C 180,E1 11832.71,E2 11832.71} C_VEL
LIN {X 0,Y 264.871,Z 741.266,A -85,B 0,C 180,E1 11829.921,E2 11829.921} C_VEL
LIN {X 0,Y 256.234,Z 754.825,A -85,B 0,C 180,E1 11826.657,E2 11826.657} C_VEL
LIN {X 0,Y 248.554,Z 766.937,A -85,B 0,C 180,E1 11822.893,E2 11822.893} C_VEL
LIN {X 0,Y 242.425,Z 777.102,A -85,B 0,C 180,E1 11818.853,E2 11818.853} C_VEL
LIN {X 0,Y 237.695,Z 785.934,A -85,B 0,C 180,E1 11814.345,E2 11814.345} C_VEL
LIN {X 0,Y 234.77,Z 792.95,A -85,B 0,C 180,E1 11809.661,E2 11809.661} C_VEL
LIN {X 0,Y 234.397,Z 794.368,A -85,B 0,C 180,E1 11808.659,E2 11808.659} C_VEL
LIN {X 0,Y 233.243,Z 803.792,A -85,B 0,C 180,E1 11804.904,E2 11804.904} C_VEL
LIN {X 0,Y 232.67,Z 811.76,A -85,B 0,C 180,E1 11800.899,E2 11800.899} C_VEL
LIN {X 0,Y 232.651,Z 817.845,A -85,B 0,C 180,E1 11796.899,E2 11796.899} C_VEL
LIN {X 0,Y 232.773,Z 821.914,A -85,B 0,C 180,E1 11793.201,E2 11793.201} C_VEL
LIN {X 0,Y 232.765,Z 824.337,A -85,B 0,C 180,E1 11789.754,E2 11789.754} C_VEL
LIN {X 0,Y 232.436,Z 825.666,A -85,B 0,C 180,E1 11785.806,E2 11785.806} C_VEL
LIN {X 0,Y 232.212,Z 825.55,A -85,B 0,C 180,E1 11781.582,E2 11781.582} C_VEL
LIN {X 0,Y 232.742,Z 823.669,A -85,B 0,C 180,E1 11776.839,E2 11776.839} C_VEL
LIN {X 0,Y 234.668,Z 819.818,A -85,B 0,C 180,E1 11771.878,E2 11771.878} C_VEL
LIN {X 0,Y 238.236,Z 814.111,A -85,B 0,C 180,E1 11767.026,E2 11767.026} C_VEL
LIN {X 0,Y 243.572,Z 806.556,A -85,B 0,C 180,E1 11762.363,E2 11762.363} C_VEL
LIN {X 0,Y 251.102,Z 796.631,A -85,B 0,C 180,E1 11757.753,E2 11757.753} C_VEL
LIN {X 0,Y 260.103,Z 785.24,A -85,B 0,C 180,E1 11753.702,E2 11753.702} C_VEL
LIN {X 0,Y 270.861,Z 771.923,A -85,B 0,C 180,E1 11750.036,E2 11750.036} C_VEL
LIN {X 0,Y 282.67,Z 757.332,A -85,B 0,C 180,E1 11746.946,E2 11746.946} C_VEL
LIN {X 0,Y 295.264,Z 741.5,A -85,B 0,C 180,E1 11744.396,E2 11744.396} C_VEL
LIN {X 0,Y 298.754,Z 737.024,A -85,B 0,C 180,E1 11743.756,E2 11743.756} C_VEL
LIN {X 0,Y 286.317,Z 751.453,A -85,B 0,C 180,E1 11741.035,E2 11741.035} C_VEL
LIN {X 0,Y 274.663,Z 764.426,A -85,B 0,C 180,E1 11737.819,E2 11737.819} C_VEL
LIN {X 0,Y 263.976,Z 775.744,A -85,B 0,C 180,E1 11734.095,E2 11734.095} C_VEL
LIN {X 0,Y 254.65,Z 785.262,A -85,B 0,C 180,E1 11729.911,E2 11729.911} C_VEL
LIN {X 0,Y 247.353,Z 792.403,A -85,B 0,C 180,E1 11725.627,E2 11725.627} C_VEL
LIN {X 0,Y 241.599,Z 797.689,A -85,B 0,C 180,E1 11721.103,E2 11721.103} C_VEL
LIN {X 0,Y 237.367,Z 801.122,A -85,B 0,C 180,E1 11716.393,E2 11716.393} C_VEL
LIN {X 0,Y 234.579,Z 802.742,A -85,B 0,C 180,E1 11711.556,E2 11711.556} C_VEL
LIN {X 0,Y 233.083,Z 802.573,A -85,B 0,C 180,E1 11706.898,E2 11706.898} C_VEL
LIN {X 0,Y 232.439,Z 800.806,A -85,B 0,C 180,E1 11702.465,E2 11702.465} C_VEL
LIN {X 0,Y 232.249,Z 797.631,A -85,B 0,C 180,E1 11698.273,E2 11698.273} C_VEL
LIN {X 0,Y 232.331,Z 792.85,A -85,B 0,C 180,E1 11694.071,E2 11694.071} C_VEL
LIN {X 0,Y 232.78,Z 786.292,A -85,B 0,C 180,E1 11689.857,E2 11689.857} C_VEL
LIN {X 0,Y 233.703,Z 778.333,A -85,B 0,C 180,E1 11685.885,E2 11685.885} C_VEL
LIN {X 0,Y 235.248,Z 768.373,A -85,B 0,C 180,E1 11681.924,E2 11681.924} C_VEL
LIN {X 0,Y 237.341,Z 756.953,A -85,B 0,C 180,E1 11678.239,E2 11678.239} C_VEL
LIN {X 0,Y 240.07,Z 743.381,A -85,B 0,C 180,E1 11674.66,E2 11674.66} C_VEL
LIN {X 0,Y 243.099,Z 728.712,A -85,B 0,C 180,E1 11671.503,E2 11671.503} C_VEL
LIN {X 0,Y 246.475,Z 711.956,A -85,B 0,C 180,E1 11668.582,E2 11668.582} C_VEL
LIN {X 0,Y 249.927,Z 693.711,A -85,B 0,C 180,E1 11666.013,E2 11666.013} C_VEL
LIN {X 0,Y 253.099,Z 675.284,A -85,B 0,C 180,E1 11663.94,E2 11663.94} C_VEL
LIN {X 0,Y 255.956,Z 655.938,A -85,B 0,C 180,E1 11662.242,E2 11662.242} C_VEL
LIN {X 0,Y 258.441,Z 635.178,A -85,B 0,C 180,E1 11660.877,E2 11660.877} C_VEL
LIN {X 0,Y 260.556,Z 611.477,A -85,B 0,C 180,E1 11659.794,E2 11659.794} C_VEL
LIN {X 0,Y 272.544,Z 476.173,A -85,B 0,C 180,E1 11654.567,E2 11654.567} C_VEL
